LIN {X 0,Y 518.643,Z 984.893,A -85,B 0,C 180,E1 13734.42,E2 13734.42} C_VEL
LIN {X 0,Y 513.947,Z 1023.237,A -85,B 0,C 180,E1 13735.843,E2 13735.843} C_VEL
LIN {X 0,Y 507.593,Z 1061.404,A -85,B 0,C 180,E1 13737.996,E2 13737.996} C_VEL
LIN {X 0,Y 500.506,Z 1096.206,A -85,B 0,C 180,E1 13740.779,E2 13740.779} C_VEL
LIN {X 0,Y 493.713,Z 1126.296,A -85,B 0,C 180,E1 13744.065,E2 13744.065} C_VEL
LIN {X 0,Y 487.682,Z 1152.198,A -85,B 0,C 180,E1 13747.868,E2 13747.868} C_VEL
LIN {X 0,Y 482.961,Z 1173.823,A -85,B 0,C 180,E1 13752.188,E2 13752.188} C_VEL
LIN {X 0,Y 479.947,Z 1190.195,A -85,B 0,C 180,E1 13756.768,E2 13756.768} C_VEL
LIN {X 0,Y 478.377,Z 1201.901,A -85,B 0,C 180,E1 13761.805,E2 13761.805} C_VEL
LIN {X 0,Y 477.916,Z 1207.569,A -85,B 0,C 180,E1 13766.365,E2 13766.365} C_VEL
LIN {X 0,Y 477.819,Z 1208.936,A -85,B 0,C 180,E1 13770,E2 13770} C_VEL
LIN {X 0,Y 477.91,Z 1207.483,A -85,B 0,C 180,E1 13773.636,E2 13773.636} C_VEL
LIN {X 0,Y 478.43,Z 1201.745,A -85,B 0,C 180,E1 13778.194,E2 13778.194} C_VEL
LIN {X 0,Y 480,Z 1189.926,A -85,B 0,C 180,E1 13783.231,E2 13783.231} C_VEL
LIN {X 0,Y 483.195,Z 1172.465,A -85,B 0,C 180,E1 13788.04,E2 13788.04} C_VEL
LIN {X 0,Y 488.136,Z 1150.333,A -85,B 0,C 180,E1 13792.351,E2 13792.351} C_VEL
LIN {X 0,Y 494.263,Z 1123.856,A -85,B 0,C 180,E1 13796.149,E2 13796.149} C_VEL
LIN {X 0,Y 501.436,Z 1091.752,A -85,B 0,C 180,E1 13799.535,E2 13799.535} C_VEL
LIN {X 0,Y 508.377,Z 1056.676,A -85,B 0,C 180,E1 13802.222,E2 13802.222} C_VEL
LIN {X 0,Y 514.491,Z 1018.573,A -85,B 0,C 180,E1 13804.271,E2 13804.271} C_VEL
LIN {X 0,Y 519.025,Z 979.497,A -85,B 0,C 180,E1 13805.64,E2 13805.64} C_VEL
LIN {X 0,Y 520.756,Z 942.856,A -85,B 0,C 180,E1 13806.431,E2 13806.431} C_VEL
LIN {X 0,Y 499.338,Z 900.262,A -85,B 0,C 180,E1 13809.238,E2 13809.238} C_VEL
LIN {X 0,Y 477.541,Z 863.723,A -85,B 0,C 180,E1 13812.378,E2 13812.378} C_VEL
LIN {X 0,Y 476.202,Z 859.31,A -85,B 0,C 180,E1 13812.759,E2 13812.759} C_VEL
LIN {X 0,Y 476.028,Z 859.31,A -85,B 0,C 180,E1 13819.816,E2 13819.816} C_VEL
LIN {X 0,Y 476.22,Z 859.31,A -85,B 0,C 180,E1 13825.823,E2 13825.823} C_VEL
LIN {X 0,Y 476.377,Z 859.31,A -85,B 0,C 180,E1 13831.513,E2 13831.513} C_VEL
LIN {X 0,Y 476.557,Z 859.31,A -85,B 0,C 180,E1 13837.579,E2 13837.579} C_VEL
LIN {X 0,Y 476.651,Z 859.31,A -85,B 0,C 180,E1 13843.382,E2 13843.382} C_VEL
LIN {X 0,Y 477.094,Z 859.31,A -85,B 0,C 180,E1 13849.929,E2 13849.929} C_VEL
LIN {X 0,Y 477.532,Z 859.31,A -85,B 0,C 180,E1 13856.365,E2 13856.365} C_VEL
LIN {X 0,Y 477.649,Z 859.31,A -85,B 0,C 180,E1 13861.82,E2 13861.82} C_VEL
LIN {X 0,Y 477.243,Z 859.31,A -85,B 0,C 180,E1 13867.297,E2 13867.297} C_VEL
LIN {X 0,Y 476.971,Z 859.31,A -85,B 0,C 180,E1 13872.848,E2 13872.848} C_VEL
LIN {X 0,Y 476.774,Z 859.31,A -85,B 0,C 180,E1 13878.529,E2 13878.529} C_VEL
LIN {X 0,Y 476.542,Z 859.31,A -85,B 0,C 180,E1 13884.412,E2 13884.412} C_VEL
LIN {X 0,Y 476.279,Z 859.31,A -85,B 0,C 180,E1 13890.794,E2 13890.794} C_VEL
LIN {X 0,Y 476.088,Z 859.31,A -85,B 0,C 180,E1 13897.278,E2 13897.278} C_VEL
LIN {X 0,Y 476.085,Z 859.334,A -85,B 0,C 180,E1 13901.129,E2 13901.129} C_VEL
LIN {X 0,Y 478.529,Z 865.012,A -85,B 0,C 180,E1 13901.556,E2 13901.556} C_VEL
LIN {X 0,Y 502.826,Z 908.11,A -85,B 0,C 180,E1 13905.163,E2 13905.163} C_VEL
LIN {X 0,Y 518.318,Z 943.312,A -85,B 0,C 180,E1 13907.539,E2 13907.539} C_VEL
LIN {X 0,Y 520.224,Z 951.642,A -85,B 0,C 180,E1 13908,E2 13908} C_VEL
LIN {X 0,Y 515.804,Z 993.529,A -85,B 0,C 180,E1 13909.437,E2 13909.437} C_VEL
LIN {X 0,Y 509.794,Z 1036.666,A -85,B 0,C 180,E1 13911.635,E2 13911.635} C_VEL
LIN {X 0,Y 502.567,Z 1078.417,A -85,B 0,C 180,E1 13914.594,E2 13914.594} C_VEL
LIN {X 0,Y 495.342,Z 1116.789,A -85,B 0,C 180,E1 13918.279,E2 13918.279} C_VEL
LIN {X 0,Y 488.813,Z 1150.319,A -85,B 0,C 180,E1 13922.541,E2 13922.541} C_VEL
LIN {X 0,Y 483.649,Z 1178.839,A -85,B 0,C 180,E1 13927.341,E2 13927.341} C_VEL
LIN {X 0,Y 480.223,Z 1201.767,A -85,B 0,C 180,E1 13932.556,E2 13932.556} C_VEL
LIN {X 0,Y 478.57,Z 1217.65,A -85,B 0,C 180,E1 13937.659,E2 13937.659} C_VEL
LIN {X 0,Y 477.922,Z 1227.864,A -85,B 0,C 180,E1 13942.714,E2 13942.714} C_VEL
LIN {X 0,Y 477.728,Z 1232.511,A -85,B 0,C 180,E1 13947.322,E2 13947.322} C_VEL
LIN {X 0,Y 475.241,Z 1233.109,A -85,B 0,C 180,E1 13948.872,E2 13948.872} C_VEL
LIN {X 0,Y 469.933,Z 1232.933,A -85,B 0,C 180,E1 13951.202,E2 13951.202} C_VEL
LIN {X 0,Y 469.852,Z 1232.873,A -85,B 0,C 180,E1 13951.471,E2 13951.471} C_VEL
LIN {X 0,Y 470.024,Z 1228.932,A -85,B 0,C 180,E1 13956.479,E2 13956.479} C_VEL
LIN {X 0,Y 470.546,Z 1219.738,A -85,B 0,C 180,E1 13961.611,E2 13961.611} C_VEL
LIN {X 0,Y 472.095,Z 1204.807,A -85,B 0,C 180,E1 13966.79,E2 13966.79} C_VEL
LIN {X 0,Y 475.116,Z 1184.672,A -85,B 0,C 180,E1 13971.762,E2 13971.762} C_VEL
LIN {X 0,Y 479.783,Z 1159.104,A -85,B 0,C 180,E1 13976.494,E2 13976.494} C_VEL
LIN {X 0,Y 486.088,Z 1127.252,A -85,B 0,C 180,E1 13980.964,E2 13980.964} C_VEL
LIN {X 0,Y 493.608,Z 1090.252,A -85,B 0,C 180,E1 13984.873,E2 13984.873} C_VEL
LIN {X 0,Y 501.082,Z 1049.955,A -85,B 0,C 180,E1 13988.053,E2 13988.053} C_VEL
LIN {X 0,Y 507.902,Z 1006.301,A -85,B 0,C 180,E1 13990.547,E2 13990.547} C_VEL
LIN {X 0,Y 513.509,Z 959.069,A -85,B 0,C 180,E1 13992.355,E2 13992.355} C_VEL
LIN {X 0,Y 513.392,Z 950.47,A -85,B 0,C 180,E1 13992.673,E2 13992.673} C_VEL
LIN {X 0,Y 500.582,Z 918.482,A -85,B 0,C 180,E1 13994.85,E2 13994.85} C_VEL
LIN {X 0,Y 477.749,Z 876.402,A -85,B 0,C 180,E1 13998.301,E2 13998.301} C_VEL
LIN {X 0,Y 468.278,Z 860.452,A -85,B 0,C 180,E1 13999.854,E2 13999.854} C_VEL
LIN {X 0,Y 468.166,Z 859.31,A -85,B 0,C 180,E1 14000.015,E2 14000.015} C_VEL
LIN {X 0,Y 468.263,Z 859.31,A -85,B 0,C 180,E1 14006.632,E2 14006.632} C_VEL
LIN {X 0,Y 468.524,Z 859.31,A -85,B 0,C 180,E1 14013.082,E2 14013.082} C_VEL
LIN {X 0,Y 468.832,Z 859.31,A -85,B 0,C 180,E1 14019.602,E2 14019.602} C_VEL
LIN {X 0,Y 468.939,Z 859.31,A -85,B 0,C 180,E1 14025.787,E2 14025.787} C_VEL
LIN {X 0,Y 469.249,Z 859.31,A -85,B 0,C 180,E1 14030.708,E2 14030.708} C_VEL
LIN {X 0,Y 469.615,Z 859.31,A -85,B 0,C 180,E1 14036.298,E2 14036.298} C_VEL
LIN {X 0,Y 469.762,Z 859.31,A -85,B 0,C 180,E1 14041.845,E2 14041.845} C_VEL
LIN {X 0,Y 469.331,Z 859.31,A -85,B 0,C 180,E1 14047.416,E2 14047.416} C_VEL
LIN {X 0,Y 469.047,Z 859.31,A -85,B 0,C 180,E1 14053.064,E2 14053.064} C_VEL
LIN {X 0,Y 468.807,Z 859.31,A -85,B 0,C 180,E1 14058.85,E2 14058.85} C_VEL
LIN {X 0,Y 468.505,Z 859.31,A -85,B 0,C 180,E1 14065.095,E2 14065.095} C_VEL
LIN {X 0,Y 468.309,Z 859.31,A -85,B 0,C 180,E1 14071.166,E2 14071.166} C_VEL
LIN {X 0,Y 468.114,Z 859.31,A -85,B 0,C 180,E1 14077.939,E2 14077.939} C_VEL
LIN {X 0,Y 468.115,Z 859.31,A -85,B 0,C 180,E1 14084.591,E2 14084.591} C_VEL
LIN {X 0,Y 468.174,Z 859.802,A -85,B 0,C 180,E1 14086.245,E2 14086.245} C_VEL
LIN {X 0,Y 470.923,Z 865.256,A -85,B 0,C 180,E1 14086.71,E2 14086.71} C_VEL
LIN {X 0,Y 495.158,Z 906.292,A -85,B 0,C 180,E1 14090.317,E2 14090.317} C_VEL
LIN {X 0,Y 515.205,Z 946.752,A -85,B 0,C 180,E1 14093.03,E2 14093.03} C_VEL
LIN {X 0,Y 512.18,Z 987.401,A -85,B 0,C 180,E1 14093.945,E2 14093.945} C_VEL
LIN {X 0,Y 507.237,Z 1025.551,A -85,B 0,C 180,E1 14095.418,E2 14095.418} C_VEL
LIN {X 0,Y 500.822,Z 1062.523,A -85,B 0,C 180,E1 14097.556,E2 14097.556} C_VEL
LIN {X 0,Y 493.611,Z 1096.638,A -85,B 0,C 180,E1 14100.33,E2 14100.33} C_VEL
LIN {X 0,Y 486.56,Z 1126.639,A -85,B 0,C 180,E1 14103.654,E2 14103.654} C_VEL
LIN {X 0,Y 480.259,Z 1152.487,A -85,B 0,C 180,E1 14107.508,E2 14107.508} C_VEL
LIN {X 0,Y 475.347,Z 1174.075,A -85,B 0,C 180,E1 14111.892,E2 14111.892} C_VEL
LIN {X 0,Y 472.183,Z 1190.422,A -85,B 0,C 180,E1 14116.546,E2 14116.546} C_VEL
LIN {X 0,Y 470.51,Z 1202.111,A -85,B 0,C 180,E1 14121.667,E2 14121.667} C_VEL
LIN {X 0,Y 470.017,Z 1207.774,A -85,B 0,C 180,E1 14126.303,E2 14126.303} C_VEL
LIN {X 0,Y 469.922,Z 1209.138,A -85,B 0,C 180,E1 14130,E2 14130} C_VEL
LIN {X 0,Y 470.013,Z 1207.688,A -85,B 0,C 180,E1 14133.697,E2 14133.697} C_VEL
LIN {X 0,Y 470.558,Z 1201.957,A -85,B 0,C 180,E1 14138.332,E2 14138.332} C_VEL
LIN {X 0,Y 472.233,Z 1190.156,A -85,B 0,C 180,E1 14143.453,E2 14143.453} C_VEL
LIN {X 0,Y 475.608,Z 1172.733,A -85,B 0,C 180,E1 14148.338,E2 14148.338} C_VEL
LIN {X 0,Y 481.056,Z 1149.238,A -85,B 0,C 180,E1 14152.943,E2 14152.943} C_VEL
LIN {X 0,Y 487.547,Z 1122.37,A -85,B 0,C 180,E1 14156.786,E2 14156.786} C_VEL
LIN {X 0,Y 494.822,Z 1090.999,A -85,B 0,C 180,E1 14160.096,E2 14160.096} C_VEL
LIN {X 0,Y 501.843,Z 1056.834,A -85,B 0,C 180,E1 14162.732,E2 14162.732} C_VEL
LIN {X 0,Y 508.188,Z 1018.409,A -85,B 0,C 180,E1 14164.819,E2 14164.819} C_VEL
LIN {X 0,Y 512.975,Z 978.573,A -85,B 0,C 180,E1 14166.213,E2 14166.213} C_VEL
LIN {X 0,Y 514.693,Z 945.644,A -85,B 0,C 180,E1 14166.937,E2 14166.937} C_VEL
LIN {X 0,Y 492.273,Z 901.174,A -85,B 0,C 180,E1 14169.979,E2 14169.979} C_VEL
LIN {X 0,Y 470.238,Z 864.606,A -85,B 0,C 180,E1 14173.277,E2 14173.277} C_VEL
LIN {X 0,Y 468.154,Z 859.31,A -85,B 0,C 180,E1 14173.753,E2 14173.753} C_VEL
LIN {X 0,Y 468.127,Z 859.31,A -85,B 0,C 180,E1 14179.672,E2 14179.672} C_VEL
LIN {X 0,Y 468.287,Z 859.31,A -85,B 0,C 180,E1 14186.64,E2 14186.64} C_VEL
LIN {X 0,Y 468.477,Z 859.31,A -85,B 0,C 180,E1 14193.085,E2 14193.085} C_VEL
LIN {X 0,Y 468.671,Z 859.31,A -85,B 0,C 180,E1 14199.656,E2 14199.656} C_VEL
LIN {X 0,Y 468.844,Z 859.31,A -85,B 0,C 180,E1 14205.836,E2 14205.836} C_VEL
LIN {X 0,Y 469.33,Z 859.31,A -85,B 0,C 180,E1 14212.227,E2 14212.227} C_VEL
LIN {X 0,Y 469.667,Z 859.31,A -85,B 0,C 180,E1 14218.154,E2 14218.154} C_VEL
LIN {X 0,Y 469.601,Z 859.31,A -85,B 0,C 180,E1 14223.702,E2 14223.702} C_VEL
LIN {X 0,Y 469.229,Z 859.31,A -85,B 0,C 180,E1 14229.292,E2 14229.292} C_VEL
LIN {X 0,Y 468.986,Z 859.31,A -85,B 0,C 180,E1 14234.978,E2 14234.978} C_VEL
LIN {X 0,Y 468.782,Z 859.31,A -85,B 0,C 180,E1 14240.825,E2 14240.825} C_VEL
LIN {X 0,Y 468.497,Z 859.31,A -85,B 0,C 180,E1 14246.919,E2 14246.919} C_VEL
LIN {X 0,Y 468.277,Z 859.31,A -85,B 0,C 180,E1 14253.367,E2 14253.367} C_VEL
LIN {X 0,Y 468.111,Z 859.312,A -85,B 0,C 180,E1 14260.118,E2 14260.118} C_VEL
LIN {X 0,Y 470.283,Z 864.719,A -85,B 0,C 180,E1 14260.525,E2 14260.525} C_VEL
LIN {X 0,Y 492.086,Z 902.116,A -85,B 0,C 180,E1 14263.914,E2 14263.914} C_VEL
LIN {X 0,Y 509.924,Z 939.992,A -85,B 0,C 180,E1 14266.663,E2 14266.663} C_VEL
LIN {X 0,Y 513.917,Z 953.77,A -85,B 0,C 180,E1 14267.504,E2 14267.504} C_VEL
LIN {X 0,Y 509.349,Z 994.883,A -85,B 0,C 180,E1 14268.95,E2 14268.95} C_VEL
LIN {X 0,Y 503.273,Z 1036.889,A -85,B 0,C 180,E1 14271.119,E2 14271.119} C_VEL
LIN {X 0,Y 495.963,Z 1077.869,A -85,B 0,C 180,E1 14274.05,E2 14274.05} C_VEL
LIN {X 0,Y 488.496,Z 1115.732,A -85,B 0,C 180,E1 14277.704,E2 14277.704} C_VEL
LIN {X 0,Y 481.527,Z 1149.949,A -85,B 0,C 180,E1 14282.089,E2 14282.089} C_VEL
LIN {X 0,Y 476.023,Z 1178.977,A -85,B 0,C 180,E1 14287.05,E2 14287.05} C_VEL
LIN {X 0,Y 472.472,Z 1201.489,A -85,B 0,C 180,E1 14292.261,E2 14292.261} C_VEL
LIN {X 0,Y 470.711,Z 1217.409,A -85,B 0,C 180,E1 14297.45,E2 14297.45} C_VEL
LIN {X 0,Y 470.105,Z 1226.204,A -85,B 0,C 180,E1 14301.66,E2 14301.66} C_VEL
LIN {X 0,Y 469.844,Z 1231.759,A -85,B 0,C 180,E1 14306.302,E2 14306.302} C_VEL
LIN {X 0,Y 469.936,Z 1233.157,A -85,B 0,C 180,E1 14310,E2 14310} C_VEL
LIN {X 0,Y 469.852,Z 1232.873,A -85,B 0,C 180,E1 14311.471,E2 14311.471} C_VEL
LIN {X 0,Y 467.415,Z 1232.232,A -85,B 0,C 180,E1 14313.044,E2 14313.044} C_VEL
LIN {X 0,Y 462.169,Z 1230.135,A -85,B 0,C 180,E1 14315.394,E2 14315.394} C_VEL
LIN {X 0,Y 462.077,Z 1229.821,A -85,B 0,C 180,E1 14315.664,E2 14315.664} C_VEL
LIN {X 0,Y 462.495,Z 1221.924,A -85,B 0,C 180,E1 14320.678,E2 14320.678} C_VEL
LIN {X 0,Y 463.939,Z 1207.878,A -85,B 0,C 180,E1 14326.085,E2 14326.085} C_VEL
LIN {X 0,Y 467.146,Z 1186.79,A -85,B 0,C 180,E1 14331.62,E2 14331.62} C_VEL
LIN {X 0,Y 472.159,Z 1160.263,A -85,B 0,C 180,E1 14336.699,E2 14336.699} C_VEL
LIN {X 0,Y 478.842,Z 1128.024,A -85,B 0,C 180,E1 14341.325,E2 14341.325} C_VEL
LIN {X 0,Y 486.665,Z 1091.024,A -85,B 0,C 180,E1 14345.307,E2 14345.307} C_VEL
LIN {X 0,Y 494.453,Z 1050.57,A -85,B 0,C 180,E1 14348.549,E2 14348.549} C_VEL
LIN {X 0,Y 501.632,Z 1006.288,A -85,B 0,C 180,E1 14351.104,E2 14351.104} C_VEL
LIN {X 0,Y 507.368,Z 959.498,A -85,B 0,C 180,E1 14352.911,E2 14352.911} C_VEL
LIN {X 0,Y 506.856,Z 951.867,A -85,B 0,C 180,E1 14353.238,E2 14353.238} C_VEL
LIN {X 0,Y 492.383,Z 916.889,A -85,B 0,C 180,E1 14355.747,E2 14355.747} C_VEL
LIN {X 0,Y 470.309,Z 876.985,A -85,B 0,C 180,E1 14359.208,E2 14359.208} C_VEL
LIN {X 0,Y 460.437,Z 860.936,A -85,B 0,C 180,E1 14360.89,E2 14360.89} C_VEL
LIN {X 0,Y 460.251,Z 859.31,A -85,B 0,C 180,E1 14361.01,E2 14361.01} C_VEL
LIN {X 0,Y 460.401,Z 859.31,A -85,B 0,C 180,E1 14368.23,E2 14368.23} C_VEL
LIN {X 0,Y 460.636,Z 859.31,A -85,B 0,C 180,E1 14374.686,E2 14374.686} C_VEL
LIN {X 0,Y 460.894,Z 859.31,A -85,B 0,C 180,E1 14380.808,E2 14380.808} C_VEL
LIN {X 0,Y 461.078,Z 859.31,A -85,B 0,C 180,E1 14386.701,E2 14386.701} C_VEL
LIN {X 0,Y 461.42,Z 859.31,A -85,B 0,C 180,E1 14392.451,E2 14392.451} C_VEL
LIN {X 0,Y 461.757,Z 859.31,A -85,B 0,C 180,E1 14398.117,E2 14398.117} C_VEL
LIN {X 0,Y 461.683,Z 859.31,A -85,B 0,C 180,E1 14403.76,E2 14403.76} C_VEL
LIN {X 0,Y 461.272,Z 859.31,A -85,B 0,C 180,E1 14409.767,E2 14409.767} C_VEL
LIN {X 0,Y 461.038,Z 859.31,A -85,B 0,C 180,E1 14415.238,E2 14415.238} C_VEL
LIN {X 0,Y 460.793,Z 859.31,A -85,B 0,C 180,E1 14421.198,E2 14421.198} C_VEL
LIN {X 0,Y 460.495,Z 859.31,A -85,B 0,C 180,E1 14427.42,E2 14427.42} C_VEL
LIN {X 0,Y 460.392,Z 859.31,A -85,B 0,C 180,E1 14431.764,E2 14431.764} C_VEL
LIN {X 0,Y 460.187,Z 859.31,A -85,B 0,C 180,E1 14438.713,E2 14438.713} C_VEL
LIN {X 0,Y 460.214,Z 859.407,A -85,B 0,C 180,E1 14445.165,E2 14445.165} C_VEL
LIN {X 0,Y 462.529,Z 864.884,A -85,B 0,C 180,E1 14445.597,E2 14445.597} C_VEL
LIN {X 0,Y 484.481,Z 900.745,A -85,B 0,C 180,E1 14449.032,E2 14449.032} C_VEL
LIN {X 0,Y 506.711,Z 944.18,A -85,B 0,C 180,E1 14452.164,E2 14452.164} C_VEL
LIN {X 0,Y 509.1,Z 950.401,A -85,B 0,C 180,E1 14452.522,E2 14452.522} C_VEL
LIN {X 0,Y 505.553,Z 991.888,A -85,B 0,C 180,E1 14453.521,E2 14453.521} C_VEL
LIN {X 0,Y 500.14,Z 1030.636,A -85,B 0,C 180,E1 14455.12,E2 14455.12} C_VEL
LIN {X 0,Y 493.483,Z 1066.438,A -85,B 0,C 180,E1 14457.302,E2 14457.302} C_VEL
LIN {X 0,Y 486.19,Z 1099.316,A -85,B 0,C 180,E1 14460.088,E2 14460.088} C_VEL
LIN {X 0,Y 478.994,Z 1128.68,A -85,B 0,C 180,E1 14463.459,E2 14463.459} C_VEL
LIN {X 0,Y 472.565,Z 1154.05,A -85,B 0,C 180,E1 14467.37,E2 14467.37} C_VEL
LIN {X 0,Y 467.733,Z 1174.324,A -85,B 0,C 180,E1 14471.587,E2 14471.587} C_VEL
LIN {X 0,Y 464.447,Z 1190.646,A -85,B 0,C 180,E1 14476.318,E2 14476.318} C_VEL
LIN {X 0,Y 462.645,Z 1202.321,A -85,B 0,C 180,E1 14481.525,E2 14481.525} C_VEL
LIN {X 0,Y 462.119,Z 1207.978,A -85,B 0,C 180,E1 14486.24,E2 14486.24} C_VEL
LIN {X 0,Y 462.039,Z 1209.339,A -85,B 0,C 180,E1 14490,E2 14490} C_VEL
LIN {X 0,Y 462.116,Z 1207.894,A -85,B 0,C 180,E1 14493.76,E2 14493.76} C_VEL
LIN {X 0,Y 462.691,Z 1202.168,A -85,B 0,C 180,E1 14498.475,E2 14498.475} C_VEL
LIN {X 0,Y 464.494,Z 1190.383,A -85,B 0,C 180,E1 14503.681,E2 14503.681} C_VEL
LIN {X 0,Y 467.779,Z 1173.951,A -85,B 0,C 180,E1 14508.411,E2 14508.411} C_VEL
LIN {X 0,Y 473.371,Z 1150.953,A -85,B 0,C 180,E1 14513.087,E2 14513.087} C_VEL
LIN {X 0,Y 480.447,Z 1122.744,A -85,B 0,C 180,E1 14517.215,E2 14517.215} C_VEL
LIN {X 0,Y 487.993,Z 1091.476,A -85,B 0,C 180,E1 14520.562,E2 14520.562} C_VEL
LIN {X 0,Y 495.345,Z 1057.016,A -85,B 0,C 180,E1 14523.253,E2 14523.253} C_VEL
LIN {X 0,Y 501.866,Z 1018.788,A -85,B 0,C 180,E1 14525.355,E2 14525.355} C_VEL
LIN {X 0,Y 506.858,Z 978.632,A -85,B 0,C 180,E1 14526.777,E2 14526.777} C_VEL
LIN {X 0,Y 508.419,Z 948.038,A -85,B 0,C 180,E1 14527.487,E2 14527.487} C_VEL
LIN {X 0,Y 487.116,Z 905.608,A -85,B 0,C 180,E1 14530.471,E2 14530.471} C_VEL
LIN {X 0,Y 465.526,Z 869.667,A -85,B 0,C 180,E1 14533.79,E2 14533.79} C_VEL
LIN {X 0,Y 460.319,Z 860.503,A -85,B 0,C 180,E1 14534.68,E2 14534.68} C_VEL
LIN {X 0,Y 460.225,Z 859.31,A -85,B 0,C 180,E1 14534.724,E2 14534.724} C_VEL
LIN {X 0,Y 460.213,Z 859.31,A -85,B 0,C 180,E1 14541.29,E2 14541.29} C_VEL
LIN {X 0,Y 460.4,Z 859.31,A -85,B 0,C 180,E1 14548.236,E2 14548.236} C_VEL
LIN {X 0,Y 460.585,Z 859.31,A -85,B 0,C 180,E1 14554.689,E2 14554.689} C_VEL
LIN {X 0,Y 460.732,Z 859.31,A -85,B 0,C 180,E1 14560.807,E2 14560.807} C_VEL
LIN {X 0,Y 461.022,Z 859.31,A -85,B 0,C 180,E1 14566.705,E2 14566.705} C_VEL
LIN {X 0,Y 461.463,Z 859.31,A -85,B 0,C 180,E1 14572.457,E2 14572.457} C_VEL
LIN {X 0,Y 461.762,Z 859.31,A -85,B 0,C 180,E1 14578.123,E2 14578.123} C_VEL
LIN {X 0,Y 461.688,Z 859.31,A -85,B 0,C 180,E1 14583.765,E2 14583.765} C_VEL
LIN {X 0,Y 461.264,Z 859.31,A -85,B 0,C 180,E1 14589.759,E2 14589.759} C_VEL
LIN {X 0,Y 461.045,Z 859.31,A -85,B 0,C 180,E1 14595.243,E2 14595.243} C_VEL
LIN {X 0,Y 460.823,Z 859.31,A -85,B 0,C 180,E1 14601.202,E2 14601.202} C_VEL
LIN {X 0,Y 460.52,Z 859.31,A -85,B 0,C 180,E1 14607.424,E2 14607.424} C_VEL
LIN {X 0,Y 460.408,Z 859.31,A -85,B 0,C 180,E1 14611.769,E2 14611.769} C_VEL
LIN {X 0,Y 460.217,Z 859.31,A -85,B 0,C 180,E1 14618.991,E2 14618.991} C_VEL
LIN {X 0,Y 462.795,Z 865.147,A -85,B 0,C 180,E1 14619.555,E2 14619.555} C_VEL
LIN {X 0,Y 484.819,Z 902.715,A -85,B 0,C 180,E1 14623.122,E2 14623.122} C_VEL
LIN {X 0,Y 502.161,Z 938.918,A -85,B 0,C 180,E1 14625.876,E2 14625.876} C_VEL
LIN {X 0,Y 507.634,Z 956.314,A -85,B 0,C 180,E1 14627.01,E2 14627.01} C_VEL
LIN {X 0,Y 502.713,Z 998.007,A -85,B 0,C 180,E1 14628.531,E2 14628.531} C_VEL
LIN {X 0,Y 496.473,Z 1038.942,A -85,B 0,C 180,E1 14630.707,E2 14630.707} C_VEL
LIN {X 0,Y 488.925,Z 1079.443,A -85,B 0,C 180,E1 14633.671,E2 14633.671} C_VEL
LIN {X 0,Y 481.158,Z 1117.321,A -85,B 0,C 180,E1 14637.415,E2 14637.415} C_VEL
LIN {X 0,Y 473.962,Z 1151.139,A -85,B 0,C 180,E1 14641.864,E2 14641.864} C_VEL
LIN {X 0,Y 468.524,Z 1178.663,A -85,B 0,C 180,E1 14646.66,E2 14646.66} C_VEL
LIN {X 0,Y 464.735,Z 1201.218,A -85,B 0,C 180,E1 14651.955,E2 14651.955} C_VEL
LIN {X 0,Y 462.873,Z 1217.171,A -85,B 0,C 180,E1 14657.234,E2 14657.234} C_VEL
LIN {X 0,Y 462.216,Z 1225.984,A -85,B 0,C 180,E1 14661.516,E2 14661.516} C_VEL
LIN {X 0,Y 461.942,Z 1231.555,A -85,B 0,C 180,E1 14666.238,E2 14666.238} C_VEL
LIN {X 0,Y 462.055,Z 1232.956,A -85,B 0,C 180,E1 14670,E2 14670} C_VEL
LIN {X 0,Y 462.003,Z 1231.559,A -85,B 0,C 180,E1 14673.761,E2 14673.761} C_VEL
LIN {X 0,Y 462.077,Z 1229.821,A -85,B 0,C 180,E1 14675.664,E2 14675.664} C_VEL
LIN {X 0,Y 460.831,Z 1228.526,A -85,B 0,C 180,E1 14676.726,E2 14676.726} C_VEL
LIN {X 0,Y 454.504,Z 1224.099,A -85,B 0,C 180,E1 14679.609,E2 14679.609} C_VEL
LIN {X 0,Y 454.462,Z 1223.629,A -85,B 0,C 180,E1 14679.881,E2 14679.881} C_VEL
LIN {X 0,Y 455.613,Z 1211.823,A -85,B 0,C 180,E1 14684.936,E2 14684.936} C_VEL
LIN {X 0,Y 458.186,Z 1193.554,A -85,B 0,C 180,E1 14690.319,E2 14690.319} C_VEL
LIN {X 0,Y 462.843,Z 1169.569,A -85,B 0,C 180,E1 14695.455,E2 14695.455} C_VEL
LIN {X 0,Y 469.331,Z 1139.313,A -85,B 0,C 180,E1 14700.296,E2 14700.296} C_VEL
LIN {X 0,Y 477.217,Z 1103.192,A -85,B 0,C 180,E1 14704.629,E2 14704.629} C_VEL
LIN {X 0,Y 485.591,Z 1063.104,A -85,B 0,C 180,E1 14708.188,E2 14708.188} C_VEL
LIN {X 0,Y 493.207,Z 1020.517,A -85,B 0,C 180,E1 14710.946,E2 14710.946} C_VEL
LIN {X 0,Y 499.618,Z 975.313,A -85,B 0,C 180,E1 14712.967,E2 14712.967} C_VEL
LIN {X 0,Y 501.077,Z 955.78,A -85,B 0,C 180,E1 14713.655,E2 14713.655} C_VEL
LIN {X 0,Y 487.368,Z 921.772,A -85,B 0,C 180,E1 14716.172,E2 14716.172} C_VEL
LIN {X 0,Y 466.105,Z 882.842,A -85,B 0,C 180,E1 14719.61,E2 14719.61} C_VEL
LIN {X 0,Y 452.501,Z 860.973,A -85,B 0,C 180,E1 14722.009,E2 14722.009} C_VEL
LIN {X 0,Y 452.314,Z 859.31,A -85,B 0,C 180,E1 14722.178,E2 14722.178} C_VEL
LIN {X 0,Y 452.388,Z 859.31,A -85,B 0,C 180,E1 14727.6,E2 14727.6} C_VEL
LIN {X 0,Y 452.669,Z 859.31,A -85,B 0,C 180,E1 14734.208,E2 14734.208} C_VEL
LIN {X 0,Y 452.941,Z 859.31,A -85,B 0,C 180,E1 14740.458,E2 14740.458} C_VEL
LIN {X 0,Y 453.14,Z 859.31,A -85,B 0,C 180,E1 14746.464,E2 14746.464} C_VEL
LIN {X 0,Y 453.51,Z 859.31,A -85,B 0,C 180,E1 14752.319,E2 14752.319} C_VEL
LIN {X 0,Y 453.875,Z 859.31,A -85,B 0,C 180,E1 14758.085,E2 14758.085} C_VEL
LIN {X 0,Y 453.778,Z 859.31,A -85,B 0,C 180,E1 14763.826,E2 14763.826} C_VEL
LIN {X 0,Y 453.403,Z 859.31,A -85,B 0,C 180,E1 14769.614,E2 14769.614} C_VEL
LIN {X 0,Y 453.111,Z 859.31,A -85,B 0,C 180,E1 14775.511,E2 14775.511} C_VEL
LIN {X 0,Y 452.855,Z 859.31,A -85,B 0,C 180,E1 14781.588,E2 14781.588} C_VEL
LIN {X 0,Y 452.52,Z 859.31,A -85,B 0,C 180,E1 14787.945,E2 14787.945} C_VEL
LIN {X 0,Y 452.337,Z 859.31,A -85,B 0,C 180,E1 14794.701,E2 14794.701} C_VEL
LIN {X 0,Y 452.218,Z 859.31,A -85,B 0,C 180,E1 14799.585,E2 14799.585} C_VEL
LIN {X 0,Y 452.293,Z 859.31,A -85,B 0,C 180,E1 14804.002,E2 14804.002} C_VEL
LIN {X 0,Y 454.772,Z 865.018,A -85,B 0,C 180,E1 14804.52,E2 14804.52} C_VEL
LIN {X 0,Y 476.117,Z 899.474,A -85,B 0,C 180,E1 14808.024,E2 14808.024} C_VEL
LIN {X 0,Y 497.352,Z 939.652,A -85,B 0,C 180,E1 14811.13,E2 14811.13} C_VEL
LIN {X 0,Y 502.965,Z 952.207,A -85,B 0,C 180,E1 14811.958,E2 14811.958} C_VEL
LIN {X 0,Y 498.971,Z 995.969,A -85,B 0,C 180,E1 14813.079,E2 14813.079} C_VEL
LIN {X 0,Y 493.057,Z 1035.538,A -85,B 0,C 180,E1 14814.814,E2 14814.814} C_VEL
LIN {X 0,Y 485.711,Z 1072.495,A -85,B 0,C 180,E1 14817.211,E2 14817.211} C_VEL
LIN {X 0,Y 477.815,Z 1105.983,A -85,B 0,C 180,E1 14820.256,E2 14820.256} C_VEL
LIN {X 0,Y 470.14,Z 1135.582,A -85,B 0,C 180,E1 14823.938,E2 14823.938} C_VEL
LIN {X 0,Y 463.631,Z 1160.578,A -85,B 0,C 180,E1 14828.175,E2 14828.175} C_VEL
LIN {X 0,Y 458.922,Z 1180.103,A -85,B 0,C 180,E1 14832.713,E2 14832.713} C_VEL
LIN {X 0,Y 455.787,Z 1195.793,A -85,B 0,C 180,E1 14838.008,E2 14838.008} C_VEL
LIN {X 0,Y 454.496,Z 1205.313,A -85,B 0,C 180,E1 14843.299,E2 14843.299} C_VEL
LIN {X 0,Y 454.136,Z 1209.215,A -85,B 0,C 180,E1 14848.088,E2 14848.088} C_VEL
LIN {X 0,Y 454.247,Z 1209.162,A -85,B 0,C 180,E1 14851.912,E2 14851.912} C_VEL
LIN {X 0,Y 454.525,Z 1205.194,A -85,B 0,C 180,E1 14856.701,E2 14856.701} C_VEL
LIN {X 0,Y 455.85,Z 1195.569,A -85,B 0,C 180,E1 14861.991,E2 14861.991} C_VEL
LIN {X 0,Y 458.951,Z 1179.773,A -85,B 0,C 180,E1 14867.287,E2 14867.287} C_VEL
LIN {X 0,Y 464.04,Z 1158.936,A -85,B 0,C 180,E1 14872.057,E2 14872.057} C_VEL
LIN {X 0,Y 470.756,Z 1133.212,A -85,B 0,C 180,E1 14876.306,E2 14876.306} C_VEL
LIN {X 0,Y 478.443,Z 1103.378,A -85,B 0,C 180,E1 14879.92,E2 14879.92} C_VEL
LIN {X 0,Y 486.284,Z 1069.61,A -85,B 0,C 180,E1 14882.911,E2 14882.911} C_VEL
LIN {X 0,Y 493.562,Z 1031.945,A -85,B 0,C 180,E1 14885.28,E2 14885.28} C_VEL
LIN {X 0,Y 499.328,Z 991.839,A -85,B 0,C 180,E1 14886.963,E2 14886.963} C_VEL
LIN {X 0,Y 502.68,Z 951.415,A -85,B 0,C 180,E1 14887.981,E2 14887.981} C_VEL
LIN {X 0,Y 480.79,Z 907.701,A -85,B 0,C 180,E1 14891.155,E2 14891.155} C_VEL
LIN {X 0,Y 458.577,Z 870.917,A -85,B 0,C 180,E1 14894.701,E2 14894.701} C_VEL
LIN {X 0,Y 452.499,Z 861.045,A -85,B 0,C 180,E1 14895.776,E2 14895.776} C_VEL
LIN {X 0,Y 452.293,Z 859.31,A -85,B 0,C 180,E1 14895.921,E2 14895.921} C_VEL
LIN {X 0,Y 452.324,Z 859.31,A -85,B 0,C 180,E1 14902.93,E2 14902.93} C_VEL
LIN {X 0,Y 452.519,Z 859.31,A -85,B 0,C 180,E1 14909.861,E2 14909.861} C_VEL
LIN {X 0,Y 452.706,Z 859.31,A -85,B 0,C 180,E1 14916.327,E2 14916.327} C_VEL
LIN {X 0,Y 452.85,Z 859.31,A -85,B 0,C 180,E1 14922.481,E2 14922.481} C_VEL
LIN {X 0,Y 453.23,Z 859.31,A -85,B 0,C 180,E1 14928.434,E2 14928.434} C_VEL
LIN {X 0,Y 453.694,Z 859.31,A -85,B 0,C 180,E1 14934.254,E2 14934.254} C_VEL
LIN {X 0,Y 454.019,Z 859.31,A -85,B 0,C 180,E1 14940.003,E2 14940.003} C_VEL
LIN {X 0,Y 453.69,Z 859.31,A -85,B 0,C 180,E1 14945.752,E2 14945.752} C_VEL
LIN {X 0,Y 453.26,Z 859.31,A -85,B 0,C 180,E1 14951.571,E2 14951.571} C_VEL
LIN {X 0,Y 453.031,Z 859.31,A -85,B 0,C 180,E1 14957.517,E2 14957.517} C_VEL
LIN {X 0,Y 452.773,Z 859.31,A -85,B 0,C 180,E1 14963.675,E2 14963.675} C_VEL
LIN {X 0,Y 452.535,Z 859.31,A -85,B 0,C 180,E1 14970.144,E2 14970.144} C_VEL
LIN {X 0,Y 452.303,Z 859.31,A -85,B 0,C 180,E1 14977.079,E2 14977.079} C_VEL
LIN {X 0,Y 452.311,Z 859.86,A -85,B 0,C 180,E1 14977.96,E2 14977.96} C_VEL
LIN {X 0,Y 455.206,Z 865.447,A -85,B 0,C 180,E1 14978.514,E2 14978.514} C_VEL
LIN {X 0,Y 477.9,Z 903.872,A -85,B 0,C 180,E1 14982.349,E2 14982.349} C_VEL
LIN {X 0,Y 495.693,Z 940.704,A -85,B 0,C 180,E1 14985.276,E2 14985.276} C_VEL
LIN {X 0,Y 501.427,Z 958.119,A -85,B 0,C 180,E1 14986.479,E2 14986.479} C_VEL
LIN {X 0,Y 496.177,Z 1000.576,A -85,B 0,C 180,E1 14988.074,E2 14988.074} C_VEL
LIN {X 0,Y 489.683,Z 1040.936,A -85,B 0,C 180,E1 14990.277,E2 14990.277} C_VEL
LIN {X 0,Y 482.109,Z 1080.122,A -85,B 0,C 180,E1 14993.202,E2 14993.202} C_VEL
LIN {X 0,Y 474.187,Z 1117.166,A -85,B 0,C 180,E1 14996.91,E2 14996.91} C_VEL
LIN {X 0,Y 466.933,Z 1150.061,A -85,B 0,C 180,E1 15001.274,E2 15001.274} C_VEL
LIN {X 0,Y 460.994,Z 1178.355,A -85,B 0,C 180,E1 15006.255,E2 15006.255} C_VEL
LIN {X 0,Y 456.998,Z 1200.95,A -85,B 0,C 180,E1 15011.639,E2 15011.639} C_VEL
LIN {X 0,Y 455.042,Z 1216.936,A -85,B 0,C 180,E1 15017.01,E2 15017.01} C_VEL
LIN {X 0,Y 454.339,Z 1225.765,A -85,B 0,C 180,E1 15021.368,E2 15021.368} C_VEL
LIN {X 0,Y 454.05,Z 1231.35,A -85,B 0,C 180,E1 15026.173,E2 15026.173} C_VEL
LIN {X 0,Y 454.156,Z 1232.754,A -85,B 0,C 180,E1 15030,E2 15030} C_VEL
LIN {X 0,Y 454.099,Z 1231.355,A -85,B 0,C 180,E1 15033.826,E2 15033.826} C_VEL
LIN {X 0,Y 454.295,Z 1225.772,A -85,B 0,C 180,E1 15038.632,E2 15038.632} C_VEL
LIN {X 0,Y 454.462,Z 1223.629,A -85,B 0,C 180,E1 15039.881,E2 15039.881} C_VEL
LIN {X 0,Y 452.246,Z 1220.571,A -85,B 0,C 180,E1 15041.471,E2 15041.471} C_VEL
LIN {X 0,Y 447.461,Z 1215.219,A -85,B 0,C 180,E1 15043.834,E2 15043.834} C_VEL
LIN {X 0,Y 447.445,Z 1214.564,A -85,B 0,C 180,E1 15044.104,E2 15044.104} C_VEL
LIN {X 0,Y 449.671,Z 1198.176,A -85,B 0,C 180,E1 15049.381,E2 15049.381} C_VEL
LIN {X 0,Y 453.689,Z 1176.83,A -85,B 0,C 180,E1 15054.413,E2 15054.413} C_VEL
LIN {X 0,Y 460.007,Z 1148.688,A -85,B 0,C 180,E1 15059.377,E2 15059.377} C_VEL
LIN {X 0,Y 467.604,Z 1115.824,A -85,B 0,C 180,E1 15063.755,E2 15063.755} C_VEL
LIN {X 0,Y 476.232,Z 1076.935,A -85,B 0,C 180,E1 15067.626,E2 15067.626} C_VEL
LIN {X 0,Y 484.45,Z 1035.521,A -85,B 0,C 180,E1 15070.647,E2 15070.647} C_VEL
LIN {X 0,Y 491.444,Z 991.551,A -85,B 0,C 180,E1 15072.927,E2 15072.927} C_VEL
LIN {X 0,Y 494.83,Z 958.061,A -85,B 0,C 180,E1 15074.195,E2 15074.195} C_VEL
LIN {X 0,Y 480.983,Z 923.85,A -85,B 0,C 180,E1 15076.836,E2 15076.836} C_VEL
LIN {X 0,Y 460.498,Z 886.612,A -85,B 0,C 180,E1 15080.261,E2 15080.261} C_VEL
LIN {X 0,Y 445.97,Z 863.98,A -85,B 0,C 180,E1 15082.904,E2 15082.904} C_VEL
LIN {X 0,Y 444.421,Z 859.31,A -85,B 0,C 180,E1 15083.269,E2 15083.269} C_VEL
LIN {X 0,Y 444.527,Z 859.31,A -85,B 0,C 180,E1 15089.254,E2 15089.254} C_VEL
LIN {X 0,Y 444.839,Z 859.31,A -85,B 0,C 180,E1 15095.877,E2 15095.877} C_VEL
LIN {X 0,Y 445.103,Z 859.31,A -85,B 0,C 180,E1 15102.405,E2 15102.405} C_VEL
LIN {X 0,Y 445.306,Z 859.31,A -85,B 0,C 180,E1 15108.22,E2 15108.22} C_VEL
LIN {X 0,Y 445.755,Z 859.31,A -85,B 0,C 180,E1 15114.146,E2 15114.146} C_VEL
LIN {X 0,Y 446.113,Z 859.31,A -85,B 0,C 180,E1 15119.997,E2 15119.997} C_VEL
LIN {X 0,Y 445.766,Z 859.31,A -85,B 0,C 180,E1 15125.849,E2 15125.849} C_VEL
LIN {X 0,Y 445.367,Z 859.31,A -85,B 0,C 180,E1 15131.773,E2 15131.773} C_VEL
LIN {X 0,Y 445.064,Z 859.31,A -85,B 0,C 180,E1 15137.836,E2 15137.836} C_VEL
LIN {X 0,Y 444.794,Z 859.31,A -85,B 0,C 180,E1 15144.12,E2 15144.12} C_VEL
LIN {X 0,Y 444.512,Z 859.31,A -85,B 0,C 180,E1 15150.741,E2 15150.741} C_VEL
LIN {X 0,Y 444.4,Z 859.31,A -85,B 0,C 180,E1 15155.412,E2 15155.412} C_VEL
LIN {X 0,Y 444.299,Z 859.31,A -85,B 0,C 180,E1 15162.775,E2 15162.775} C_VEL
LIN {X 0,Y 446.783,Z 865.028,A -85,B 0,C 180,E1 15163.343,E2 15163.343} C_VEL
LIN {X 0,Y 468.403,Z 899.119,A -85,B 0,C 180,E1 15167.063,E2 15167.063} C_VEL
LIN {X 0,Y 489.396,Z 938.343,A -85,B 0,C 180,E1 15170.262,E2 15170.262} C_VEL
LIN {X 0,Y 496.897,Z 955.689,A -85,B 0,C 180,E1 15171.431,E2 15171.431} C_VEL
LIN {X 0,Y 492.733,Z 997.104,A -85,B 0,C 180,E1 15172.532,E2 15172.532} C_VEL
LIN {X 0,Y 486.648,Z 1036.249,A -85,B 0,C 180,E1 15174.28,E2 15174.28} C_VEL
LIN {X 0,Y 478.965,Z 1073.475,A -85,B 0,C 180,E1 15176.737,E2 15176.737} C_VEL
LIN {X 0,Y 470.849,Z 1106.688,A -85,B 0,C 180,E1 15179.813,E2 15179.813} C_VEL
LIN {X 0,Y 462.976,Z 1135.969,A -85,B 0,C 180,E1 15183.517,E2 15183.517} C_VEL
LIN {X 0,Y 456.228,Z 1160.842,A -85,B 0,C 180,E1 15187.803,E2 15187.803} C_VEL
LIN {X 0,Y 451.306,Z 1180.339,A -85,B 0,C 180,E1 15192.412,E2 15192.412} C_VEL
LIN {X 0,Y 448,Z 1196.01,A -85,B 0,C 180,E1 15197.796,E2 15197.796} C_VEL
LIN {X 0,Y 446.63,Z 1205.518,A -85,B 0,C 180,E1 15203.181,E2 15203.181} C_VEL
LIN {X 0,Y 446.237,Z 1209.417,A -85,B 0,C 180,E1 15208.054,E2 15208.054} C_VEL
LIN {X 0,Y 446.345,Z 1209.365,A -85,B 0,C 180,E1 15211.946,E2 15211.946} C_VEL
LIN {X 0,Y 446.661,Z 1205.401,A -85,B 0,C 180,E1 15216.819,E2 15216.819} C_VEL
LIN {X 0,Y 448.052,Z 1195.788,A -85,B 0,C 180,E1 15222.203,E2 15222.203} C_VEL
LIN {X 0,Y 451.327,Z 1180.012,A -85,B 0,C 180,E1 15227.588,E2 15227.588} C_VEL
LIN {X 0,Y 456.652,Z 1159.216,A -85,B 0,C 180,E1 15232.433,E2 15232.433} C_VEL
LIN {X 0,Y 463.581,Z 1133.786,A -85,B 0,C 180,E1 15236.708,E2 15236.708} C_VEL
LIN {X 0,Y 471.866,Z 1102.628,A -85,B 0,C 180,E1 15240.52,E2 15240.52} C_VEL
LIN {X 0,Y 479.996,Z 1068.642,A -85,B 0,C 180,E1 15243.536,E2 15243.536} C_VEL
LIN {X 0,Y 487.344,Z 1031.714,A -85,B 0,C 180,E1 15245.867,E2 15245.867} C_VEL
LIN {X 0,Y 493.294,Z 991.671,A -85,B 0,C 180,E1 15247.557,E2 15247.557} C_VEL
LIN {X 0,Y 496.376,Z 953.617,A -85,B 0,C 180,E1 15248.572,E2 15248.572} C_VEL
LIN {X 0,Y 475.792,Z 912.254,A -85,B 0,C 180,E1 15251.66,E2 15251.66} C_VEL
LIN {X 0,Y 454.318,Z 876.463,A -85,B 0,C 180,E1 15255.18,E2 15255.18} C_VEL
LIN {X 0,Y 446.027,Z 864.188,A -85,B 0,C 180,E1 15256.672,E2 15256.672} C_VEL
LIN {X 0,Y 444.303,Z 859.31,A -85,B 0,C 180,E1 15257.117,E2 15257.117} C_VEL
LIN {X 0,Y 444.31,Z 859.31,A -85,B 0,C 180,E1 15262.145,E2 15262.145} C_VEL
LIN {X 0,Y 444.482,Z 859.31,A -85,B 0,C 180,E1 15268.461,E2 15268.461} C_VEL
LIN {X 0,Y 444.642,Z 859.31,A -85,B 0,C 180,E1 15273.713,E2 15273.713} C_VEL
LIN {X 0,Y 444.872,Z 859.31,A -85,B 0,C 180,E1 15280.094,E2 15280.094} C_VEL
LIN {X 0,Y 445.157,Z 859.31,A -85,B 0,C 180,E1 15286.222,E2 15286.222} C_VEL
LIN {X 0,Y 445.622,Z 859.31,A -85,B 0,C 180,E1 15292.263,E2 15292.263} C_VEL
LIN {X 0,Y 445.972,Z 859.31,A -85,B 0,C 180,E1 15298.056,E2 15298.056} C_VEL
LIN {X 0,Y 445.87,Z 859.31,A -85,B 0,C 180,E1 15303.899,E2 15303.899} C_VEL
LIN {X 0,Y 445.474,Z 859.31,A -85,B 0,C 180,E1 15309.792,E2 15309.792} C_VEL
LIN {X 0,Y 445.157,Z 859.31,A -85,B 0,C 180,E1 15315.801,E2 15315.801} C_VEL
LIN {X 0,Y 444.919,Z 859.31,A -85,B 0,C 180,E1 15321.998,E2 15321.998} C_VEL
LIN {X 0,Y 444.615,Z 859.31,A -85,B 0,C 180,E1 15328.493,E2 15328.493} C_VEL
LIN {X 0,Y 444.406,Z 859.31,A -85,B 0,C 180,E1 15335.418,E2 15335.418} C_VEL
LIN {X 0,Y 444.457,Z 859.732,A -85,B 0,C 180,E1 15336.782,E2 15336.782} C_VEL
LIN {X 0,Y 446.801,Z 864.966,A -85,B 0,C 180,E1 15337.277,E2 15337.277} C_VEL
LIN {X 0,Y 468.062,Z 899.737,A -85,B 0,C 180,E1 15341.056,E2 15341.056} C_VEL
LIN {X 0,Y 487.036,Z 937.387,A -85,B 0,C 180,E1 15344.255,E2 15344.255} C_VEL
LIN {X 0,Y 495.219,Z 960.393,A -85,B 0,C 180,E1 15345.948,E2 15345.948} C_VEL
LIN {X 0,Y 489.436,Z 1004.601,A -85,B 0,C 180,E1 15347.669,E2 15347.669} C_VEL
LIN {X 0,Y 482.369,Z 1046.057,A -85,B 0,C 180,E1 15350.043,E2 15350.043} C_VEL
LIN {X 0,Y 474.451,Z 1084.783,A -85,B 0,C 180,E1 15353.079,E2 15353.079} C_VEL
LIN {X 0,Y 466.616,Z 1119.884,A -85,B 0,C 180,E1 15356.741,E2 15356.741} C_VEL
LIN {X 0,Y 459.46,Z 1150.959,A -85,B 0,C 180,E1 15360.981,E2 15360.981} C_VEL
LIN {X 0,Y 453.261,Z 1179.239,A -85,B 0,C 180,E1 15366.087,E2 15366.087} C_VEL
LIN {X 0,Y 449.197,Z 1201.197,A -85,B 0,C 180,E1 15371.452,E2 15371.452} C_VEL
LIN {X 0,Y 447.19,Z 1216.702,A -85,B 0,C 180,E1 15376.778,E2 15376.778} C_VEL
LIN {X 0,Y 446.472,Z 1225.548,A -85,B 0,C 180,E1 15381.215,E2 15381.215} C_VEL
LIN {X 0,Y 446.148,Z 1231.146,A -85,B 0,C 180,E1 15386.105,E2 15386.105} C_VEL
LIN {X 0,Y 446.258,Z 1232.552,A -85,B 0,C 180,E1 15390,E2 15390} C_VEL
LIN {X 0,Y 446.196,Z 1231.151,A -85,B 0,C 180,E1 15393.894,E2 15393.894} C_VEL
LIN {X 0,Y 446.428,Z 1225.556,A -85,B 0,C 180,E1 15398.786,E2 15398.786} C_VEL
LIN {X 0,Y 447.445,Z 1214.564,A -85,B 0,C 180,E1 15404.104,E2 15404.104} C_VEL
LIN {X 0,Y 444.206,Z 1209.081,A -85,B 0,C 180,E1 15406.204,E2 15406.204} C_VEL
LIN {X 0,Y 441.209,Z 1202.872,A -85,B 0,C 180,E1 15408.302,E2 15408.302} C_VEL
LIN {X 0,Y 445.262,Z 1181.411,A -85,B 0,C 180,E1 15413.799,E2 15413.799} C_VEL
LIN {X 0,Y 451.067,Z 1155.367,A -85,B 0,C 180,E1 15418.759,E2 15418.759} C_VEL
LIN {X 0,Y 458.344,Z 1125.712,A -85,B 0,C 180,E1 15423.058,E2 15423.058} C_VEL
LIN {X 0,Y 466.834,Z 1089.552,A -85,B 0,C 180,E1 15427.046,E2 15427.046} C_VEL
LIN {X 0,Y 475.18,Z 1050.786,A -85,B 0,C 180,E1 15430.232,E2 15430.232} C_VEL
LIN {X 0,Y 482.982,Z 1007.264,A -85,B 0,C 180,E1 15432.816,E2 15432.816} C_VEL
LIN {X 0,Y 488.834,Z 961.104,A -85,B 0,C 180,E1 15434.694,E2 15434.694} C_VEL
LIN {X 0,Y 475.063,Z 926.733,A -85,B 0,C 180,E1 15437.45,E2 15437.45} C_VEL
LIN {X 0,Y 454.125,Z 888.629,A -85,B 0,C 180,E1 15441.086,E2 15441.086} C_VEL
LIN {X 0,Y 438.411,Z 864.45,A -85,B 0,C 180,E1 15444.075,E2 15444.075} C_VEL
LIN {X 0,Y 436.514,Z 859.31,A -85,B 0,C 180,E1 15444.64,E2 15444.64} C_VEL
LIN {X 0,Y 436.645,Z 859.31,A -85,B 0,C 180,E1 15450.938,E2 15450.938} C_VEL
LIN {X 0,Y 437.011,Z 859.31,A -85,B 0,C 180,E1 15457.582,E2 15457.582} C_VEL
LIN {X 0,Y 437.192,Z 859.31,A -85,B 0,C 180,E1 15463.904,E2 15463.904} C_VEL
LIN {X 0,Y 437.54,Z 859.31,A -85,B 0,C 180,E1 15470.028,E2 15470.028} C_VEL
LIN {X 0,Y 437.979,Z 859.31,A -85,B 0,C 180,E1 15476.031,E2 15476.031} C_VEL
LIN {X 0,Y 438.154,Z 859.31,A -85,B 0,C 180,E1 15481.979,E2 15481.979} C_VEL
LIN {X 0,Y 437.656,Z 859.31,A -85,B 0,C 180,E1 15487.956,E2 15487.956} C_VEL
LIN {X 0,Y 437.326,Z 859.31,A -85,B 0,C 180,E1 15494.03,E2 15494.03} C_VEL
LIN {X 0,Y 437.034,Z 859.31,A -85,B 0,C 180,E1 15500.586,E2 15500.586} C_VEL
LIN {X 0,Y 436.693,Z 859.31,A -85,B 0,C 180,E1 15506.803,E2 15506.803} C_VEL
LIN {X 0,Y 436.477,Z 859.31,A -85,B 0,C 180,E1 15513.729,E2 15513.729} C_VEL
LIN {X 0,Y 436.312,Z 859.31,A -85,B 0,C 180,E1 15520.178,E2 15520.178} C_VEL
LIN {X 0,Y 436.384,Z 860.08,A -85,B 0,C 180,E1 15521.58,E2 15521.58} C_VEL
LIN {X 0,Y 439.281,Z 865.428,A -85,B 0,C 180,E1 15522.18,E2 15522.18} C_VEL
LIN {X 0,Y 461.903,Z 901.01,A -85,B 0,C 180,E1 15526.259,E2 15526.259} C_VEL
LIN {X 0,Y 482.443,Z 938.937,A -85,B 0,C 180,E1 15529.503,E2 15529.503} C_VEL
LIN {X 0,Y 490.836,Z 957.605,A -85,B 0,C 180,E1 15530.857,E2 15530.857} C_VEL
LIN {X 0,Y 486.551,Z 998.21,A -85,B 0,C 180,E1 15531.971,E2 15531.971} C_VEL
LIN {X 0,Y 480.57,Z 1035.568,A -85,B 0,C 180,E1 15533.655,E2 15533.655} C_VEL
LIN {X 0,Y 472.925,Z 1071.786,A -85,B 0,C 180,E1 15536.035,E2 15536.035} C_VEL
LIN {X 0,Y 464.315,Z 1106.034,A -85,B 0,C 180,E1 15539.206,E2 15539.206} C_VEL
LIN {X 0,Y 455.864,Z 1136.276,A -85,B 0,C 180,E1 15543.071,E2 15543.071} C_VEL
LIN {X 0,Y 448.811,Z 1161.106,A -85,B 0,C 180,E1 15547.416,E2 15547.416} C_VEL
LIN {X 0,Y 443.664,Z 1180.573,A -85,B 0,C 180,E1 15552.098,E2 15552.098} C_VEL
LIN {X 0,Y 440.418,Z 1195.127,A -85,B 0,C 180,E1 15557.077,E2 15557.077} C_VEL
LIN {X 0,Y 438.869,Z 1204.426,A -85,B 0,C 180,E1 15562.062,E2 15562.062} C_VEL
LIN {X 0,Y 438.453,Z 1208.59,A -85,B 0,C 180,E1 15566.037,E2 15566.037} C_VEL
LIN {X 0,Y 438.379,Z 1209.944,A -85,B 0,C 180,E1 15570,E2 15570} C_VEL
LIN {X 0,Y 438.455,Z 1208.507,A -85,B 0,C 180,E1 15573.964,E2 15573.964} C_VEL
LIN {X 0,Y 439.126,Z 1202.799,A -85,B 0,C 180,E1 15578.933,E2 15578.933} C_VEL
LIN {X 0,Y 441.267,Z 1191.057,A -85,B 0,C 180,E1 15584.416,E2 15584.416} C_VEL
LIN {X 0,Y 445.607,Z 1172.736,A -85,B 0,C 180,E1 15589.88,E2 15589.88} C_VEL
LIN {X 0,Y 451.71,Z 1150.621,A -85,B 0,C 180,E1 15594.496,E2 15594.496} C_VEL
LIN {X 0,Y 459.334,Z 1123.839,A -85,B 0,C 180,E1 15598.577,E2 15598.577} C_VEL
LIN {X 0,Y 467.981,Z 1091.639,A -85,B 0,C 180,E1 15602.157,E2 15602.157} C_VEL
LIN {X 0,Y 476.174,Z 1056.909,A -85,B 0,C 180,E1 15604.946,E2 15604.946} C_VEL
LIN {X 0,Y 483.27,Z 1019.631,A -85,B 0,C 180,E1 15607.054,E2 15607.054} C_VEL
LIN {X 0,Y 488.793,Z 979.229,A -85,B 0,C 180,E1 15608.538,E2 15608.538} C_VEL
LIN {X 0,Y 490.175,Z 956.01,A -85,B 0,C 180,E1 15609.152,E2 15609.152} C_VEL
LIN {X 0,Y 470.5,Z 916.251,A -85,B 0,C 180,E1 15612.226,E2 15612.226} C_VEL
LIN {X 0,Y 449.949,Z 881.764,A -85,B 0,C 180,E1 15615.695,E2 15615.695} C_VEL
LIN {X 0,Y 438.435,Z 864.609,A -85,B 0,C 180,E1 15617.85,E2 15617.85} C_VEL
LIN {X 0,Y 436.335,Z 859.31,A -85,B 0,C 180,E1 15618.477,E2 15618.477} C_VEL
LIN {X 0,Y 436.399,Z 859.31,A -85,B 0,C 180,E1 15623.837,E2 15623.837} C_VEL
LIN {X 0,Y 436.583,Z 859.31,A -85,B 0,C 180,E1 15630.193,E2 15630.193} C_VEL
LIN {X 0,Y 436.789,Z 859.31,A -85,B 0,C 180,E1 15635.409,E2 15635.409} C_VEL
LIN {X 0,Y 436.978,Z 859.31,A -85,B 0,C 180,E1 15641.823,E2 15641.823} C_VEL
LIN {X 0,Y 437.346,Z 859.31,A -85,B 0,C 180,E1 15648.008,E2 15648.008} C_VEL
LIN {X 0,Y 437.849,Z 859.31,A -85,B 0,C 180,E1 15654.045,E2 15654.045} C_VEL
LIN {X 0,Y 438.231,Z 859.31,A -85,B 0,C 180,E1 15660.003,E2 15660.003} C_VEL
LIN {X 0,Y 437.838,Z 859.31,A -85,B 0,C 180,E1 15665.961,E2 15665.961} C_VEL
LIN {X 0,Y 437.392,Z 859.31,A -85,B 0,C 180,E1 15671.997,E2 15671.997} C_VEL
LIN {X 0,Y 437.133,Z 859.31,A -85,B 0,C 180,E1 15678.176,E2 15678.176} C_VEL
LIN {X 0,Y 436.835,Z 859.31,A -85,B 0,C 180,E1 15684.594,E2 15684.594} C_VEL
LIN {X 0,Y 436.609,Z 859.31,A -85,B 0,C 180,E1 15691.366,E2 15691.366} C_VEL
LIN {X 0,Y 436.536,Z 859.31,A -85,B 0,C 180,E1 15695.486,E2 15695.486} C_VEL
LIN {X 0,Y 438.873,Z 864.902,A -85,B 0,C 180,E1 15696.04,E2 15696.04} C_VEL
LIN {X 0,Y 460.425,Z 899.428,A -85,B 0,C 180,E1 15700.061,E2 15700.061} C_VEL
LIN {X 0,Y 479.857,Z 937.483,A -85,B 0,C 180,E1 15703.461,E2 15703.461} C_VEL
LIN {X 0,Y 489.056,Z 962.27,A -85,B 0,C 180,E1 15705.398,E2 15705.398} C_VEL
LIN {X 0,Y 482.89,Z 1007.357,A -85,B 0,C 180,E1 15707.195,E2 15707.195} C_VEL
LIN {X 0,Y 475.242,Z 1050.401,A -85,B 0,C 180,E1 15709.753,E2 15709.753} C_VEL
LIN {X 0,Y 466.628,Z 1090.582,A -85,B 0,C 180,E1 15713.063,E2 15713.063} C_VEL
LIN {X 0,Y 457.717,Z 1128.069,A -85,B 0,C 180,E1 15717.241,E2 15717.241} C_VEL
LIN {X 0,Y 449.939,Z 1160.294,A -85,B 0,C 180,E1 15722.07,E2 15722.07} C_VEL
LIN {X 0,Y 444.285,Z 1186.859,A -85,B 0,C 180,E1 15727.433,E2 15727.433} C_VEL
LIN {X 0,Y 440.603,Z 1206.991,A -85,B 0,C 180,E1 15733.002,E2 15733.002} C_VEL
LIN {X 0,Y 439.028,Z 1219.841,A -85,B 0,C 180,E1 15738.048,E2 15738.048} C_VEL
LIN {X 0,Y 438.471,Z 1228.08,A -85,B 0,C 180,E1 15743.053,E2 15743.053} C_VEL
LIN {X 0,Y 438.364,Z 1231.993,A -85,B 0,C 180,E1 15748.019,E2 15748.019} C_VEL
LIN {X 0,Y 438.327,Z 1231.993,A -85,B 0,C 180,E1 15751.981,E2 15751.981} C_VEL
LIN {X 0,Y 438.459,Z 1228.088,A -85,B 0,C 180,E1 15756.947,E2 15756.947} C_VEL
LIN {X 0,Y 439.148,Z 1218.838,A -85,B 0,C 180,E1 15762.454,E2 15762.454} C_VEL
LIN {X 0,Y 441.059,Z 1203.797,A -85,B 0,C 180,E1 15768.011,E2 15768.011} C_VEL
LIN {X 0,Y 441.209,Z 1202.872,A -85,B 0,C 180,E1 15768.302,E2 15768.302} C_VEL
LIN {X 0,Y 438.588,Z 1196.147,A -85,B 0,C 180,E1 15770.382,E2 15770.382} C_VEL
LIN {X 0,Y 436.261,Z 1188.736,A -85,B 0,C 180,E1 15772.447,E2 15772.447} C_VEL
LIN {X 0,Y 441.592,Z 1165.092,A -85,B 0,C 180,E1 15777.485,E2 15777.485} C_VEL
LIN {X 0,Y 448.766,Z 1135.73,A -85,B 0,C 180,E1 15782.233,E2 15782.233} C_VEL
LIN {X 0,Y 457.193,Z 1102.436,A -85,B 0,C 180,E1 15786.305,E2 15786.305} C_VEL
LIN {X 0,Y 465.92,Z 1064.433,A -85,B 0,C 180,E1 15789.813,E2 15789.813} C_VEL
LIN {X 0,Y 474.518,Z 1021.385,A -85,B 0,C 180,E1 15792.688,E2 15792.688} C_VEL
LIN {X 0,Y 481.519,Z 976.753,A -85,B 0,C 180,E1 15794.738,E2 15794.738} C_VEL
LIN {X 0,Y 482.491,Z 962.811,A -85,B 0,C 180,E1 15795.293,E2 15795.293} C_VEL
LIN {X 0,Y 468.217,Z 927.63,A -85,B 0,C 180,E1 15798.253,E2 15798.253} C_VEL
LIN {X 0,Y 448.475,Z 892.092,A -85,B 0,C 180,E1 15801.808,E2 15801.808} C_VEL
LIN {X 0,Y 430.975,Z 864.957,A -85,B 0,C 180,E1 15805.3,E2 15805.3} C_VEL
LIN {X 0,Y 428.59,Z 859.31,A -85,B 0,C 180,E1 15806.01,E2 15806.01} C_VEL
LIN {X 0,Y 428.767,Z 859.31,A -85,B 0,C 180,E1 15812.655,E2 15812.655} C_VEL
LIN {X 0,Y 429.143,Z 859.31,A -85,B 0,C 180,E1 15819.326,E2 15819.326} C_VEL
LIN {X 0,Y 429.352,Z 859.31,A -85,B 0,C 180,E1 15825.698,E2 15825.698} C_VEL
LIN {X 0,Y 429.734,Z 859.31,A -85,B 0,C 180,E1 15831.891,E2 15831.891} C_VEL
LIN {X 0,Y 430.161,Z 859.31,A -85,B 0,C 180,E1 15837.979,E2 15837.979} C_VEL
LIN {X 0,Y 430.053,Z 859.31,A -85,B 0,C 180,E1 15844.037,E2 15844.037} C_VEL
LIN {X 0,Y 429.627,Z 859.31,A -85,B 0,C 180,E1 15850.152,E2 15850.152} C_VEL
LIN {X 0,Y 429.272,Z 859.31,A -85,B 0,C 180,E1 15856.396,E2 15856.396} C_VEL
LIN {X 0,Y 428.923,Z 859.31,A -85,B 0,C 180,E1 15863.289,E2 15863.289} C_VEL
LIN {X 0,Y 428.692,Z 859.31,A -85,B 0,C 180,E1 15869.648,E2 15869.648} C_VEL
LIN {X 0,Y 428.447,Z 859.31,A -85,B 0,C 180,E1 15876.944,E2 15876.944} C_VEL
LIN {X 0,Y 428.412,Z 859.461,A -85,B 0,C 180,E1 15880.2,E2 15880.2} C_VEL
LIN {X 0,Y 430.783,Z 864.945,A -85,B 0,C 180,E1 15880.753,E2 15880.753} C_VEL
LIN {X 0,Y 448.789,Z 892.004,A -85,B 0,C 180,E1 15884.245,E2 15884.245} C_VEL
LIN {X 0,Y 470.285,Z 929.285,A -85,B 0,C 180,E1 15887.889,E2 15887.889} C_VEL
LIN {X 0,Y 484.793,Z 960.6,A -85,B 0,C 180,E1 15890.296,E2 15890.296} C_VEL
LIN {X 0,Y 480.194,Z 1000.732,A -85,B 0,C 180,E1 15891.448,E2 15891.448} C_VEL
LIN {X 0,Y 473.857,Z 1038.244,A -85,B 0,C 180,E1 15893.205,E2 15893.205} C_VEL
LIN {X 0,Y 466.069,Z 1073.634,A -85,B 0,C 180,E1 15895.605,E2 15895.605} C_VEL
LIN {X 0,Y 457.501,Z 1106.409,A -85,B 0,C 180,E1 15898.696,E2 15898.696} C_VEL
LIN {X 0,Y 449.232,Z 1135.029,A -85,B 0,C 180,E1 15902.368,E2 15902.368} C_VEL
LIN {X 0,Y 441.78,Z 1160.208,A -85,B 0,C 180,E1 15906.769,E2 15906.769} C_VEL
LIN {X 0,Y 436.072,Z 1180.805,A -85,B 0,C 180,E1 15911.776,E2 15911.776} C_VEL
LIN {X 0,Y 432.648,Z 1195.346,A -85,B 0,C 180,E1 15916.841,E2 15916.841} C_VEL
LIN {X 0,Y 431.001,Z 1204.635,A -85,B 0,C 180,E1 15921.916,E2 15921.916} C_VEL
LIN {X 0,Y 430.556,Z 1208.794,A -85,B 0,C 180,E1 15925.964,E2 15925.964} C_VEL
LIN {X 0,Y 430.481,Z 1210.146,A -85,B 0,C 180,E1 15930,E2 15930} C_VEL
LIN {X 0,Y 430.559,Z 1208.712,A -85,B 0,C 180,E1 15934.036,E2 15934.036} C_VEL
LIN {X 0,Y 431.282,Z 1203.008,A -85,B 0,C 180,E1 15939.097,E2 15939.097} C_VEL
LIN {X 0,Y 433.563,Z 1191.278,A -85,B 0,C 180,E1 15944.678,E2 15944.678} C_VEL
LIN {X 0,Y 438.095,Z 1172.992,A -85,B 0,C 180,E1 15950.236,E2 15950.236} C_VEL
LIN {X 0,Y 444.687,Z 1150.156,A -85,B 0,C 180,E1 15955.054,E2 15955.054} C_VEL
LIN {X 0,Y 452.893,Z 1122.202,A -85,B 0,C 180,E1 15959.315,E2 15959.315} C_VEL
LIN {X 0,Y 461.729,Z 1090.436,A -85,B 0,C 180,E1 15962.833,E2 15962.833} C_VEL
LIN {X 0,Y 470.13,Z 1055.9,A -85,B 0,C 180,E1 15965.6,E2 15965.6} C_VEL
LIN {X 0,Y 477.44,Z 1018.098,A -85,B 0,C 180,E1 15967.731,E2 15967.731} C_VEL
LIN {X 0,Y 482.904,Z 978.95,A -85,B 0,C 180,E1 15969.168,E2 15969.168} C_VEL
LIN {X 0,Y 484.292,Z 959.041,A -85,B 0,C 180,E1 15969.695,E2 15969.695} C_VEL
LIN {X 0,Y 465.077,Z 919.803,A -85,B 0,C 180,E1 15972.837,E2 15972.837} C_VEL
LIN {X 0,Y 443.55,Z 883.524,A -85,B 0,C 180,E1 15976.61,E2 15976.61} C_VEL
LIN {X 0,Y 430.551,Z 864.719,A -85,B 0,C 180,E1 15979.167,E2 15979.167} C_VEL
LIN {X 0,Y 428.428,Z 859.31,A -85,B 0,C 180,E1 15979.702,E2 15979.702} C_VEL
LIN {X 0,Y 428.483,Z 859.31,A -85,B 0,C 180,E1 15985.554,E2 15985.554} C_VEL
LIN {X 0,Y 428.702,Z 859.31,A -85,B 0,C 180,E1 15992.087,E2 15992.087} C_VEL
LIN {X 0,Y 428.923,Z 859.31,A -85,B 0,C 180,E1 15997.142,E2 15997.142} C_VEL
LIN {X 0,Y 429.101,Z 859.31,A -85,B 0,C 180,E1 16003.598,E2 16003.598} C_VEL
LIN {X 0,Y 429.64,Z 859.31,A -85,B 0,C 180,E1 16009.849,E2 16009.849} C_VEL
LIN {X 0,Y 430.069,Z 859.31,A -85,B 0,C 180,E1 16015.963,E2 16015.963} C_VEL
LIN {X 0,Y 430.248,Z 859.31,A -85,B 0,C 180,E1 16022.021,E2 16022.021} C_VEL
LIN {X 0,Y 429.719,Z 859.31,A -85,B 0,C 180,E1 16028.109,E2 16028.109} C_VEL
LIN {X 0,Y 429.392,Z 859.31,A -85,B 0,C 180,E1 16034.3,E2 16034.3} C_VEL
LIN {X 0,Y 429.144,Z 859.31,A -85,B 0,C 180,E1 16040.674,E2 16040.674} C_VEL
LIN {X 0,Y 428.736,Z 859.31,A -85,B 0,C 180,E1 16047.348,E2 16047.348} C_VEL
LIN {X 0,Y 428.605,Z 859.31,A -85,B 0,C 180,E1 16054.153,E2 16054.153} C_VEL
LIN {X 0,Y 430.852,Z 864.824,A -85,B 0,C 180,E1 16054.711,E2 16054.711} C_VEL
LIN {X 0,Y 448.295,Z 891.911,A -85,B 0,C 180,E1 16058.188,E2 16058.188} C_VEL
LIN {X 0,Y 468.045,Z 927.559,A -85,B 0,C 180,E1 16061.745,E2 16061.745} C_VEL
LIN {X 0,Y 482.114,Z 961.932,A -85,B 0,C 180,E1 16064.641,E2 16064.641} C_VEL
LIN {X 0,Y 482.387,Z 968.01,A -85,B 0,C 180,E1 16064.958,E2 16064.958} C_VEL
LIN {X 0,Y 476.538,Z 1009.111,A -85,B 0,C 180,E1 16066.672,E2 16066.672} C_VEL
LIN {X 0,Y 468.639,Z 1051.802,A -85,B 0,C 180,E1 16069.258,E2 16069.258} C_VEL
LIN {X 0,Y 459.698,Z 1091.903,A -85,B 0,C 180,E1 16072.627,E2 16072.627} C_VEL
LIN {X 0,Y 451.009,Z 1127.217,A -85,B 0,C 180,E1 16076.621,E2 16076.621} C_VEL
LIN {X 0,Y 442.639,Z 1160.351,A -85,B 0,C 180,E1 16081.642,E2 16081.642} C_VEL
LIN {X 0,Y 436.712,Z 1186.581,A -85,B 0,C 180,E1 16087.019,E2 16087.019} C_VEL
LIN {X 0,Y 432.841,Z 1206.743,A -85,B 0,C 180,E1 16092.688,E2 16092.688} C_VEL
LIN {X 0,Y 431.099,Z 1220.635,A -85,B 0,C 180,E1 16098.339,E2 16098.339} C_VEL
LIN {X 0,Y 430.516,Z 1229.01,A -85,B 0,C 180,E1 16103.939,E2 16103.939} C_VEL
LIN {X 0,Y 430.458,Z 1231.791,A -85,B 0,C 180,E1 16107.982,E2 16107.982} C_VEL
LIN {X 0,Y 430.423,Z 1231.791,A -85,B 0,C 180,E1 16112.017,E2 16112.017} C_VEL
LIN {X 0,Y 430.55,Z 1227.878,A -85,B 0,C 180,E1 16117.075,E2 16117.075} C_VEL
LIN {X 0,Y 431.323,Z 1218.617,A -85,B 0,C 180,E1 16122.684,E2 16122.684} C_VEL
LIN {X 0,Y 433.355,Z 1203.395,A -85,B 0,C 180,E1 16128.394,E2 16128.394} C_VEL
LIN {X 0,Y 436.261,Z 1188.736,A -85,B 0,C 180,E1 16132.447,E2 16132.447} C_VEL
LIN {X 0,Y 434.156,Z 1180.87,A -85,B 0,C 180,E1 16134.491,E2 16134.491} C_VEL
LIN {X 0,Y 432.452,Z 1172.346,A -85,B 0,C 180,E1 16136.505,E2 16136.505} C_VEL
LIN {X 0,Y 439.489,Z 1144.787,A -85,B 0,C 180,E1 16141.395,E2 16141.395} C_VEL
LIN {X 0,Y 447.704,Z 1112.965,A -85,B 0,C 180,E1 16145.695,E2 16145.695} C_VEL
LIN {X 0,Y 456.994,Z 1075.679,A -85,B 0,C 180,E1 16149.471,E2 16149.471} C_VEL
LIN {X 0,Y 465.775,Z 1035.639,A -85,B 0,C 180,E1 16152.458,E2 16152.458} C_VEL
LIN {X 0,Y 473.43,Z 992.155,A -85,B 0,C 180,E1 16154.76,E2 16154.76} C_VEL
LIN {X 0,Y 476.362,Z 965.581,A -85,B 0,C 180,E1 16155.838,E2 16155.838} C_VEL
LIN {X 0,Y 462.719,Z 931.212,A -85,B 0,C 180,E1 16158.839,E2 16158.839} C_VEL
LIN {X 0,Y 442.782,Z 894.965,A -85,B 0,C 180,E1 16162.58,E2 16162.58} C_VEL
LIN {X 0,Y 423.579,Z 865.404,A -85,B 0,C 180,E1 16166.597,E2 16166.597} C_VEL
LIN {X 0,Y 420.849,Z 860.952,A -85,B 0,C 180,E1 16167.237,E2 16167.237} C_VEL
LIN {X 0,Y 420.678,Z 859.31,A -85,B 0,C 180,E1 16167.445,E2 16167.445} C_VEL
LIN {X 0,Y 420.915,Z 859.31,A -85,B 0,C 180,E1 16174.41,E2 16174.41} C_VEL
LIN {X 0,Y 421.227,Z 859.31,A -85,B 0,C 180,E1 16181.112,E2 16181.112} C_VEL
LIN {X 0,Y 421.508,Z 859.31,A -85,B 0,C 180,E1 16187.544,E2 16187.544} C_VEL
LIN {X 0,Y 422.008,Z 859.31,A -85,B 0,C 180,E1 16193.815,E2 16193.815} C_VEL
LIN {X 0,Y 422.434,Z 859.31,A -85,B 0,C 180,E1 16199.997,E2 16199.997} C_VEL
LIN {X 0,Y 422.014,Z 859.31,A -85,B 0,C 180,E1 16206.179,E2 16206.179} C_VEL
LIN {X 0,Y 421.557,Z 859.31,A -85,B 0,C 180,E1 16212.449,E2 16212.449} C_VEL
LIN {X 0,Y 421.215,Z 859.31,A -85,B 0,C 180,E1 16218.883,E2 16218.883} C_VEL
LIN {X 0,Y 420.844,Z 859.31,A -85,B 0,C 180,E1 16225.823,E2 16225.823} C_VEL
LIN {X 0,Y 420.587,Z 859.31,A -85,B 0,C 180,E1 16232.699,E2 16232.699} C_VEL
LIN {X 0,Y 420.544,Z 859.31,A -85,B 0,C 180,E1 16238.728,E2 16238.728} C_VEL
LIN {X 0,Y 422.834,Z 864.9,A -85,B 0,C 180,E1 16239.331,E2 16239.331} C_VEL
LIN {X 0,Y 440.765,Z 891.307,A -85,B 0,C 180,E1 16243.018,E2 16243.018} C_VEL
LIN {X 0,Y 461.266,Z 926.143,A -85,B 0,C 180,E1 16246.686,E2 16246.686} C_VEL
LIN {X 0,Y 478.7,Z 962.704,A -85,B 0,C 180,E1 16249.685,E2 16249.685} C_VEL
LIN {X 0,Y 473.873,Z 1003.242,A -85,B 0,C 180,E1 16250.91,E2 16250.91} C_VEL
LIN {X 0,Y 467.224,Z 1040.661,A -85,B 0,C 180,E1 16252.728,E2 16252.728} C_VEL
LIN {X 0,Y 459.197,Z 1075.492,A -85,B 0,C 180,E1 16255.16,E2 16255.16} C_VEL
LIN {X 0,Y 450.426,Z 1107.808,A -85,B 0,C 180,E1 16258.289,E2 16258.289} C_VEL
LIN {X 0,Y 441.705,Z 1136.883,A -85,B 0,C 180,E1 16262.134,E2 16262.134} C_VEL
LIN {X 0,Y 434.065,Z 1161.626,A -85,B 0,C 180,E1 16266.604,E2 16266.604} C_VEL
LIN {X 0,Y 428.484,Z 1181.037,A -85,B 0,C 180,E1 16271.442,E2 16271.442} C_VEL
LIN {X 0,Y 424.888,Z 1195.562,A -85,B 0,C 180,E1 16276.597,E2 16276.597} C_VEL
LIN {X 0,Y 423.155,Z 1204.842,A -85,B 0,C 180,E1 16281.765,E2 16281.765} C_VEL
LIN {X 0,Y 422.676,Z 1208.997,A -85,B 0,C 180,E1 16285.889,E2 16285.889} C_VEL
LIN {X 0,Y 422.608,Z 1210.347,A -85,B 0,C 180,E1 16290,E2 16290} C_VEL
LIN {X 0,Y 422.68,Z 1208.916,A -85,B 0,C 180,E1 16294.112,E2 16294.112} C_VEL
LIN {X 0,Y 423.427,Z 1203.217,A -85,B 0,C 180,E1 16299.267,E2 16299.267} C_VEL
LIN {X 0,Y 425.844,Z 1191.5,A -85,B 0,C 180,E1 16304.95,E2 16304.95} C_VEL
LIN {X 0,Y 430.625,Z 1173.245,A -85,B 0,C 180,E1 16310.603,E2 16310.603} C_VEL
LIN {X 0,Y 437.665,Z 1149.766,A -85,B 0,C 180,E1 16315.617,E2 16315.617} C_VEL
LIN {X 0,Y 445.854,Z 1123.003,A -85,B 0,C 180,E1 16319.757,E2 16319.757} C_VEL
LIN {X 0,Y 455.093,Z 1090.882,A -85,B 0,C 180,E1 16323.375,E2 16323.375} C_VEL
LIN {X 0,Y 463.696,Z 1056.771,A -85,B 0,C 180,E1 16326.15,E2 16326.15} C_VEL
LIN {X 0,Y 471.27,Z 1019.043,A -85,B 0,C 180,E1 16328.313,E2 16328.313} C_VEL
LIN {X 0,Y 477.076,Z 978.948,A -85,B 0,C 180,E1 16329.803,E2 16329.803} C_VEL
LIN {X 0,Y 478.2,Z 961.584,A -85,B 0,C 180,E1 16330.295,E2 16330.295} C_VEL
LIN {X 0,Y 459.732,Z 923.456,A -85,B 0,C 180,E1 16333.455,E2 16333.455} C_VEL
LIN {X 0,Y 439.135,Z 888.729,A -85,B 0,C 180,E1 16337.173,E2 16337.173} C_VEL
LIN {X 0,Y 423.051,Z 865.093,A -85,B 0,C 180,E1 16340.489,E2 16340.489} C_VEL
LIN {X 0,Y 420.592,Z 859.767,A -85,B 0,C 180,E1 16341.091,E2 16341.091} C_VEL
LIN {X 0,Y 420.597,Z 859.31,A -85,B 0,C 180,E1 16347.302,E2 16347.302} C_VEL
LIN {X 0,Y 420.86,Z 859.31,A -85,B 0,C 180,E1 16354.412,E2 16354.412} C_VEL
LIN {X 0,Y 421.093,Z 859.31,A -85,B 0,C 180,E1 16361.111,E2 16361.111} C_VEL
LIN {X 0,Y 421.472,Z 859.31,A -85,B 0,C 180,E1 16367.549,E2 16367.549} C_VEL
LIN {X 0,Y 422.028,Z 859.31,A -85,B 0,C 180,E1 16373.821,E2 16373.821} C_VEL
LIN {X 0,Y 422.438,Z 859.31,A -85,B 0,C 180,E1 16380.003,E2 16380.003} C_VEL
LIN {X 0,Y 422.012,Z 859.31,A -85,B 0,C 180,E1 16386.185,E2 16386.185} C_VEL
LIN {X 0,Y 421.533,Z 859.31,A -85,B 0,C 180,E1 16392.455,E2 16392.455} C_VEL
LIN {X 0,Y 421.234,Z 859.31,A -85,B 0,C 180,E1 16398.888,E2 16398.888} C_VEL
LIN {X 0,Y 420.894,Z 859.31,A -85,B 0,C 180,E1 16405.592,E2 16405.592} C_VEL
LIN {X 0,Y 420.709,Z 859.31,A -85,B 0,C 180,E1 16412.695,E2 16412.695} C_VEL
LIN {X 0,Y 422.926,Z 864.821,A -85,B 0,C 180,E1 16413.302,E2 16413.302} C_VEL
LIN {X 0,Y 430.144,Z 875.435,A -85,B 0,C 180,E1 16414.89,E2 16414.89} C_VEL
LIN {X 0,Y 450.349,Z 908.094,A -85,B 0,C 180,E1 16418.892,E2 16418.892} C_VEL
LIN {X 0,Y 468.503,Z 944.38,A -85,B 0,C 180,E1 16422.362,E2 16422.362} C_VEL
LIN {X 0,Y 476.628,Z 967.451,A -85,B 0,C 180,E1 16424.3,E2 16424.3} C_VEL
LIN {X 0,Y 470.452,Z 1009.51,A -85,B 0,C 180,E1 16426.061,E2 16426.061} C_VEL
LIN {X 0,Y 462.524,Z 1051.133,A -85,B 0,C 180,E1 16428.595,E2 16428.595} C_VEL
LIN {X 0,Y 453.388,Z 1090.673,A -85,B 0,C 180,E1 16431.922,E2 16431.922} C_VEL
LIN {X 0,Y 444.193,Z 1126.826,A -85,B 0,C 180,E1 16436.04,E2 16436.04} C_VEL
LIN {X 0,Y 435.831,Z 1158.56,A -85,B 0,C 180,E1 16440.872,E2 16440.872} C_VEL
LIN {X 0,Y 429.383,Z 1185.187,A -85,B 0,C 180,E1 16446.331,E2 16446.331} C_VEL
LIN {X 0,Y 425.359,Z 1204.891,A -85,B 0,C 180,E1 16451.837,E2 16451.837} C_VEL
LIN {X 0,Y 423.49,Z 1218.382,A -85,B 0,C 180,E1 16457.077,E2 16457.077} C_VEL
LIN {X 0,Y 422.686,Z 1227.659,A -85,B 0,C 180,E1 16462.792,E2 16462.792} C_VEL
LIN {X 0,Y 422.568,Z 1231.589,A -85,B 0,C 180,E1 16467.945,E2 16467.945} C_VEL
LIN {X 0,Y 422.54,Z 1231.589,A -85,B 0,C 180,E1 16472.055,E2 16472.055} C_VEL
LIN {X 0,Y 422.67,Z 1227.669,A -85,B 0,C 180,E1 16477.208,E2 16477.208} C_VEL
LIN {X 0,Y 423.502,Z 1218.398,A -85,B 0,C 180,E1 16482.922,E2 16482.922} C_VEL
LIN {X 0,Y 425.628,Z 1203.309,A -85,B 0,C 180,E1 16488.688,E2 16488.688} C_VEL
LIN {X 0,Y 429.685,Z 1183.727,A -85,B 0,C 180,E1 16494.015,E2 16494.015} C_VEL
LIN {X 0,Y 432.452,Z 1172.346,A -85,B 0,C 180,E1 16496.505,E2 16496.505} C_VEL
LIN {X 0,Y 431.04,Z 1163.37,A -85,B 0,C 180,E1 16498.493,E2 16498.493} C_VEL
LIN {X 0,Y 429.657,Z 1155.094,A -85,B 0,C 180,E1 16500.209,E2 16500.209} C_VEL
LIN {X 0,Y 429.949,Z 1153.772,A -85,B 0,C 180,E1 16500.44,E2 16500.44} C_VEL
LIN {X 0,Y 437.938,Z 1124.559,A -85,B 0,C 180,E1 16504.813,E2 16504.813} C_VEL
LIN {X 0,Y 447.231,Z 1089.311,A -85,B 0,C 180,E1 16508.82,E2 16508.82} C_VEL
LIN {X 0,Y 456.463,Z 1050.71,A -85,B 0,C 180,E1 16512.079,E2 16512.079} C_VEL
LIN {X 0,Y 465.01,Z 1007.136,A -85,B 0,C 180,E1 16514.722,E2 16514.722} C_VEL
LIN {X 0,Y 470.334,Z 968.519,A -85,B 0,C 180,E1 16516.383,E2 16516.383} C_VEL
LIN {X 0,Y 457.173,Z 934.775,A -85,B 0,C 180,E1 16519.432,E2 16519.432} C_VEL
LIN {X 0,Y 438.487,Z 900.379,A -85,B 0,C 180,E1 16523.098,E2 16523.098} C_VEL
LIN {X 0,Y 419.964,Z 871.697,A -85,B 0,C 180,E1 16527.079,E2 16527.079} C_VEL
LIN {X 0,Y 415.133,Z 864.887,A -85,B 0,C 180,E1 16528.224,E2 16528.224} C_VEL
LIN {X 0,Y 412.866,Z 860.37,A -85,B 0,C 180,E1 16528.823,E2 16528.823} C_VEL
LIN {X 0,Y 412.797,Z 859.31,A -85,B 0,C 180,E1 16529.081,E2 16529.081} C_VEL
LIN {X 0,Y 413.179,Z 859.31,A -85,B 0,C 180,E1 16536.469,E2 16536.469} C_VEL
LIN {X 0,Y 413.384,Z 859.31,A -85,B 0,C 180,E1 16542.949,E2 16542.949} C_VEL
LIN {X 0,Y 413.72,Z 859.31,A -85,B 0,C 180,E1 16549.448,E2 16549.448} C_VEL
LIN {X 0,Y 414.257,Z 859.31,A -85,B 0,C 180,E1 16555.803,E2 16555.803} C_VEL
LIN {X 0,Y 414.44,Z 859.31,A -85,B 0,C 180,E1 16562.092,E2 16562.092} C_VEL
LIN {X 0,Y 413.851,Z 859.31,A -85,B 0,C 180,E1 16568.665,E2 16568.665} C_VEL
LIN {X 0,Y 413.499,Z 859.31,A -85,B 0,C 180,E1 16574.857,E2 16574.857} C_VEL
LIN {X 0,Y 413.185,Z 859.31,A -85,B 0,C 180,E1 16581.505,E2 16581.505} C_VEL
LIN {X 0,Y 412.843,Z 859.31,A -85,B 0,C 180,E1 16588.488,E2 16588.488} C_VEL
LIN {X 0,Y 412.654,Z 859.31,A -85,B 0,C 180,E1 16593.409,E2 16593.409} C_VEL
LIN {X 0,Y 412.582,Z 859.872,A -85,B 0,C 180,E1 16597.196,E2 16597.196} C_VEL
LIN {X 0,Y 415.367,Z 865.327,A -85,B 0,C 180,E1 16597.913,E2 16597.913} C_VEL
LIN {X 0,Y 433.177,Z 891.26,A -85,B 0,C 180,E1 16601.804,E2 16601.804} C_VEL
LIN {X 0,Y 453.724,Z 925.758,A -85,B 0,C 180,E1 16605.668,E2 16605.668} C_VEL
LIN {X 0,Y 471.471,Z 962.269,A -85,B 0,C 180,E1 16608.839,E2 16608.839} C_VEL
LIN {X 0,Y 472.59,Z 968.11,A -85,B 0,C 180,E1 16609.163,E2 16609.163} C_VEL
LIN {X 0,Y 466.952,Z 1009.63,A -85,B 0,C 180,E1 16610.519,E2 16610.519} C_VEL
LIN {X 0,Y 459.602,Z 1047.755,A -85,B 0,C 180,E1 16612.522,E2 16612.522} C_VEL
LIN {X 0,Y 450.511,Z 1084.409,A -85,B 0,C 180,E1 16615.319,E2 16615.319} C_VEL
LIN {X 0,Y 441.26,Z 1116.249,A -85,B 0,C 180,E1 16618.709,E2 16618.709} C_VEL
LIN {X 0,Y 432.161,Z 1144.802,A -85,B 0,C 180,E1 16622.882,E2 16622.882} C_VEL
LIN {X 0,Y 425.09,Z 1167.243,A -85,B 0,C 180,E1 16627.368,E2 16627.368} C_VEL
LIN {X 0,Y 419.476,Z 1186.232,A -85,B 0,C 180,E1 16632.662,E2 16632.662} C_VEL
LIN {X 0,Y 416.206,Z 1200.059,A -85,B 0,C 180,E1 16638.449,E2 16638.449} C_VEL
LIN {X 0,Y 414.975,Z 1207.481,A -85,B 0,C 180,E1 16643.711,E2 16643.711} C_VEL
LIN {X 0,Y 414.664,Z 1210.226,A -85,B 0,C 180,E1 16647.906,E2 16647.906} C_VEL
LIN {X 0,Y 414.74,Z 1210.177,A -85,B 0,C 180,E1 16652.094,E2 16652.094} C_VEL
LIN {X 0,Y 415.164,Z 1206.226,A -85,B 0,C 180,E1 16657.34,E2 16657.34} C_VEL
LIN {X 0,Y 416.932,Z 1196.656,A -85,B 0,C 180,E1 16663.13,E2 16663.13} C_VEL
LIN {X 0,Y 420.936,Z 1180.952,A -85,B 0,C 180,E1 16668.904,E2 16668.904} C_VEL
LIN {X 0,Y 427.595,Z 1159.062,A -85,B 0,C 180,E1 16674.328,E2 16674.328} C_VEL
LIN {X 0,Y 435.797,Z 1133.417,A -85,B 0,C 180,E1 16678.845,E2 16678.845} C_VEL
LIN {X 0,Y 445.41,Z 1102.071,A -85,B 0,C 180,E1 16682.834,E2 16682.834} C_VEL
LIN {X 0,Y 454.712,Z 1067.851,A -85,B 0,C 180,E1 16685.969,E2 16685.969} C_VEL
LIN {X 0,Y 462.992,Z 1030.976,A -85,B 0,C 180,E1 16688.358,E2 16688.358} C_VEL
LIN {X 0,Y 469.579,Z 992.129,A -85,B 0,C 180,E1 16690.044,E2 16690.044} C_VEL
LIN {X 0,Y 472.363,Z 964.535,A -85,B 0,C 180,E1 16690.874,E2 16690.874} C_VEL
LIN {X 0,Y 454.785,Z 927.784,A -85,B 0,C 180,E1 16694.026,E2 16694.026} C_VEL
LIN {X 0,Y 434.686,Z 893.756,A -85,B 0,C 180,E1 16697.766,E2 16697.766} C_VEL
LIN {X 0,Y 415.542,Z 865.401,A -85,B 0,C 180,E1 16701.916,E2 16701.916} C_VEL
LIN {X 0,Y 412.679,Z 860.372,A -85,B 0,C 180,E1 16702.634,E2 16702.634} C_VEL
LIN {X 0,Y 412.573,Z 859.31,A -85,B 0,C 180,E1 16702.798,E2 16702.798} C_VEL
LIN {X 0,Y 412.715,Z 859.31,A -85,B 0,C 180,E1 16709.081,E2 16709.081} C_VEL
LIN {X 0,Y 413.028,Z 859.31,A -85,B 0,C 180,E1 16716.209,E2 16716.209} C_VEL
LIN {X 0,Y 413.22,Z 859.31,A -85,B 0,C 180,E1 16722.948,E2 16722.948} C_VEL
LIN {X 0,Y 413.775,Z 859.31,A -85,B 0,C 180,E1 16729.455,E2 16729.455} C_VEL
LIN {X 0,Y 414.264,Z 859.31,A -85,B 0,C 180,E1 16735.809,E2 16735.809} C_VEL
LIN {X 0,Y 414.445,Z 859.31,A -85,B 0,C 180,E1 16742.098,E2 16742.098} C_VEL
LIN {X 0,Y 413.841,Z 859.31,A -85,B 0,C 180,E1 16748.653,E2 16748.653} C_VEL
LIN {X 0,Y 413.508,Z 859.31,A -85,B 0,C 180,E1 16754.862,E2 16754.862} C_VEL
LIN {X 0,Y 413.216,Z 859.31,A -85,B 0,C 180,E1 16761.51,E2 16761.51} C_VEL
LIN {X 0,Y 412.867,Z 859.31,A -85,B 0,C 180,E1 16768.493,E2 16768.493} C_VEL
LIN {X 0,Y 412.764,Z 859.734,A -85,B 0,C 180,E1 16771.182,E2 16771.182} C_VEL
LIN {X 0,Y 415.225,Z 865.068,A -85,B 0,C 180,E1 16771.844,E2 16771.844} C_VEL
LIN {X 0,Y 425.513,Z 879.842,A -85,B 0,C 180,E1 16774.211,E2 16774.211} C_VEL
LIN {X 0,Y 447.304,Z 915.618,A -85,B 0,C 180,E1 16778.647,E2 16778.647} C_VEL
LIN {X 0,Y 464.278,Z 951.615,A -85,B 0,C 180,E1 16782.143,E2 16782.143} C_VEL
LIN {X 0,Y 470.499,Z 969.982,A -85,B 0,C 180,E1 16783.727,E2 16783.727} C_VEL
LIN {X 0,Y 464.175,Z 1011.277,A -85,B 0,C 180,E1 16785.506,E2 16785.506} C_VEL
LIN {X 0,Y 456.103,Z 1052.12,A -85,B 0,C 180,E1 16788.04,E2 16788.04} C_VEL
LIN {X 0,Y 446.722,Z 1091.239,A -85,B 0,C 180,E1 16791.377,E2 16791.377} C_VEL
LIN {X 0,Y 437.404,Z 1126.44,A -85,B 0,C 180,E1 16795.439,E2 16795.439} C_VEL
LIN {X 0,Y 428.694,Z 1158.24,A -85,B 0,C 180,E1 16800.34,E2 16800.34} C_VEL
LIN {X 0,Y 422.151,Z 1183.785,A -85,B 0,C 180,E1 16805.62,E2 16805.62} C_VEL
LIN {X 0,Y 417.934,Z 1203.04,A -85,B 0,C 180,E1 16810.955,E2 16810.955} C_VEL
LIN {X 0,Y 415.653,Z 1218.161,A -85,B 0,C 180,E1 16816.829,E2 16816.829} C_VEL
LIN {X 0,Y 414.791,Z 1227.449,A -85,B 0,C 180,E1 16822.654,E2 16822.654} C_VEL
LIN {X 0,Y 414.661,Z 1231.386,A -85,B 0,C 180,E1 16827.906,E2 16827.906} C_VEL
LIN {X 0,Y 414.635,Z 1231.387,A -85,B 0,C 180,E1 16832.094,E2 16832.094} C_VEL
LIN {X 0,Y 414.773,Z 1227.46,A -85,B 0,C 180,E1 16837.346,E2 16837.346} C_VEL
LIN {X 0,Y 415.667,Z 1218.179,A -85,B 0,C 180,E1 16843.17,E2 16843.17} C_VEL
LIN {X 0,Y 417.916,Z 1203.069,A -85,B 0,C 180,E1 16849.046,E2 16849.046} C_VEL
LIN {X 0,Y 422.119,Z 1183.824,A -85,B 0,C 180,E1 16854.382,E2 16854.382} C_VEL
LIN {X 0,Y 428.62,Z 1158.306,A -85,B 0,C 180,E1 16859.665,E2 16859.665} C_VEL
LIN {X 0,Y 429.949,Z 1153.772,A -85,B 0,C 180,E1 16860.44,E2 16860.44} C_VEL
LIN {X 0,Y 429.14,Z 1143.722,A -85,B 0,C 180,E1 16862.355,E2 16862.355} C_VEL
LIN {X 0,Y 428.358,Z 1134.543,A -85,B 0,C 180,E1 16863.995,E2 16863.995} C_VEL
LIN {X 0,Y 428.744,Z 1133.07,A -85,B 0,C 180,E1 16864.208,E2 16864.208} C_VEL
LIN {X 0,Y 437.955,Z 1099.849,A -85,B 0,C 180,E1 16868.346,E2 16868.346} C_VEL
LIN {X 0,Y 447.362,Z 1063.132,A -85,B 0,C 180,E1 16871.78,E2 16871.78} C_VEL
LIN {X 0,Y 456.633,Z 1020.682,A -85,B 0,C 180,E1 16874.658,E2 16874.658} C_VEL
LIN {X 0,Y 464.208,Z 975.89,A -85,B 0,C 180,E1 16876.736,E2 16876.736} C_VEL
LIN {X 0,Y 464.028,Z 970.383,A -85,B 0,C 180,E1 16877.036,E2 16877.036} C_VEL
LIN {X 0,Y 451.164,Z 937.28,A -85,B 0,C 180,E1 16880.151,E2 16880.151} C_VEL
LIN {X 0,Y 433.401,Z 904.381,A -85,B 0,C 180,E1 16883.8,E2 16883.8} C_VEL
LIN {X 0,Y 415.534,Z 876.766,A -85,B 0,C 180,E1 16887.774,E2 16887.774} C_VEL
LIN {X 0,Y 407.737,Z 865.418,A -85,B 0,C 180,E1 16889.729,E2 16889.729} C_VEL
LIN {X 0,Y 405.026,Z 860.923,A -85,B 0,C 180,E1 16890.469,E2 16890.469} C_VEL
LIN {X 0,Y 404.883,Z 859.31,A -85,B 0,C 180,E1 16890.718,E2 16890.718} C_VEL
LIN {X 0,Y 405.138,Z 859.31,A -85,B 0,C 180,E1 16895.71,E2 16895.71} C_VEL
LIN {X 0,Y 405.45,Z 859.31,A -85,B 0,C 180,E1 16902.605,E2 16902.605} C_VEL
LIN {X 0,Y 405.779,Z 859.31,A -85,B 0,C 180,E1 16909.239,E2 16909.239} C_VEL
LIN {X 0,Y 406.337,Z 859.31,A -85,B 0,C 180,E1 16915.721,E2 16915.721} C_VEL
LIN {X 0,Y 406.531,Z 859.31,A -85,B 0,C 180,E1 16922.133,E2 16922.133} C_VEL
LIN {X 0,Y 405.98,Z 859.31,A -85,B 0,C 180,E1 16928.581,E2 16928.581} C_VEL
LIN {X 0,Y 405.557,Z 859.31,A -85,B 0,C 180,E1 16935.154,E2 16935.154} C_VEL
LIN {X 0,Y 405.224,Z 859.31,A -85,B 0,C 180,E1 16941.949,E2 16941.949} C_VEL
LIN {X 0,Y 404.838,Z 859.31,A -85,B 0,C 180,E1 16949.105,E2 16949.105} C_VEL
LIN {X 0,Y 404.602,Z 859.31,A -85,B 0,C 180,E1 16955.465,E2 16955.465} C_VEL
LIN {X 0,Y 406.606,Z 864.53,A -85,B 0,C 180,E1 16956.071,E2 16956.071} C_VEL
LIN {X 0,Y 409.714,Z 868.238,A -85,B 0,C 180,E1 16956.843,E2 16956.843} C_VEL
LIN {X 0,Y 429.51,Z 897.377,A -85,B 0,C 180,E1 16961.342,E2 16961.342} C_VEL
LIN {X 0,Y 449.563,Z 931.39,A -85,B 0,C 180,E1 16965.21,E2 16965.21} C_VEL
LIN {X 0,Y 466.229,Z 966.683,A -85,B 0,C 180,E1 16968.355,E2 16968.355} C_VEL
LIN {X 0,Y 466.003,Z 976.351,A -85,B 0,C 180,E1 16968.713,E2 16968.713} C_VEL
LIN {X 0,Y 459.934,Z 1016.609,A -85,B 0,C 180,E1 16970.18,E2 16970.18} C_VEL
LIN {X 0,Y 452.269,Z 1053.093,A -85,B 0,C 180,E1 16972.234,E2 16972.234} C_VEL
LIN {X 0,Y 443.453,Z 1086.853,A -85,B 0,C 180,E1 16974.928,E2 16974.928} C_VEL
LIN {X 0,Y 434.474,Z 1116.588,A -85,B 0,C 180,E1 16978.163,E2 16978.163} C_VEL
LIN {X 0,Y 425.063,Z 1145.082,A -85,B 0,C 180,E1 16982.391,E2 16982.391} C_VEL
LIN {X 0,Y 417.393,Z 1168.471,A -85,B 0,C 180,E1 16987.192,E2 16987.192} C_VEL
LIN {X 0,Y 411.868,Z 1186.454,A -85,B 0,C 180,E1 16992.331,E2 16992.331} C_VEL
LIN {X 0,Y 408.394,Z 1200.269,A -85,B 0,C 180,E1 16998.225,E2 16998.225} C_VEL
LIN {X 0,Y 407.097,Z 1207.686,A -85,B 0,C 180,E1 17003.589,E2 17003.589} C_VEL
LIN {X 0,Y 406.778,Z 1210.428,A -85,B 0,C 180,E1 17007.865,E2 17007.865} C_VEL
LIN {X 0,Y 406.845,Z 1210.379,A -85,B 0,C 180,E1 17012.135,E2 17012.135} C_VEL
LIN {X 0,Y 407.289,Z 1206.432,A -85,B 0,C 180,E1 17017.482,E2 17017.482} C_VEL
LIN {X 0,Y 409.161,Z 1196.872,A -85,B 0,C 180,E1 17023.384,E2 17023.384} C_VEL
LIN {X 0,Y 412.844,Z 1182.848,A -85,B 0,C 180,E1 17028.733,E2 17028.733} C_VEL
LIN {X 0,Y 419.135,Z 1162.863,A -85,B 0,C 180,E1 17033.999,E2 17033.999} C_VEL
LIN {X 0,Y 427.263,Z 1138.456,A -85,B 0,C 180,E1 17038.606,E2 17038.606} C_VEL
LIN {X 0,Y 436.533,Z 1109.835,A -85,B 0,C 180,E1 17042.55,E2 17042.55} C_VEL
LIN {X 0,Y 445.773,Z 1078.182,A -85,B 0,C 180,E1 17045.75,E2 17045.75} C_VEL
LIN {X 0,Y 454.561,Z 1042.729,A -85,B 0,C 180,E1 17048.331,E2 17048.331} C_VEL
LIN {X 0,Y 461.893,Z 1004.778,A -85,B 0,C 180,E1 17050.231,E2 17050.231} C_VEL
LIN {X 0,Y 466.377,Z 967.287,A -85,B 0,C 180,E1 17051.49,E2 17051.49} C_VEL
LIN {X 0,Y 449.725,Z 931.815,A -85,B 0,C 180,E1 17054.639,E2 17054.639} C_VEL
LIN {X 0,Y 429.864,Z 897.904,A -85,B 0,C 180,E1 17058.464,E2 17058.464} C_VEL
LIN {X 0,Y 411.654,Z 871.234,A -85,B 0,C 180,E1 17062.533,E2 17062.533} C_VEL
LIN {X 0,Y 407.464,Z 865.363,A -85,B 0,C 180,E1 17063.575,E2 17063.575} C_VEL
LIN {X 0,Y 404.714,Z 860.425,A -85,B 0,C 180,E1 17064.324,E2 17064.324} C_VEL
LIN {X 0,Y 404.635,Z 859.31,A -85,B 0,C 180,E1 17064.389,E2 17064.389} C_VEL
LIN {X 0,Y 404.843,Z 859.31,A -85,B 0,C 180,E1 17070.896,E2 17070.896} C_VEL
LIN {X 0,Y 405.044,Z 859.31,A -85,B 0,C 180,E1 17075.71,E2 17075.71} C_VEL
LIN {X 0,Y 405.307,Z 859.31,A -85,B 0,C 180,E1 17082.605,E2 17082.605} C_VEL
LIN {X 0,Y 405.823,Z 859.31,A -85,B 0,C 180,E1 17089.246,E2 17089.246} C_VEL
LIN {X 0,Y 406.345,Z 859.31,A -85,B 0,C 180,E1 17095.727,E2 17095.727} C_VEL
LIN {X 0,Y 406.536,Z 859.31,A -85,B 0,C 180,E1 17102.138,E2 17102.138} C_VEL
LIN {X 0,Y 405.969,Z 859.31,A -85,B 0,C 180,E1 17108.587,E2 17108.587} C_VEL
LIN {X 0,Y 405.566,Z 859.31,A -85,B 0,C 180,E1 17115.16,E2 17115.16} C_VEL
LIN {X 0,Y 405.275,Z 859.31,A -85,B 0,C 180,E1 17121.953,E2 17121.953} C_VEL
LIN {X 0,Y 404.868,Z 859.31,A -85,B 0,C 180,E1 17129.109,E2 17129.109} C_VEL
LIN {X 0,Y 404.856,Z 859.685,A -85,B 0,C 180,E1 17129.498,E2 17129.498} C_VEL
LIN {X 0,Y 407.026,Z 864.794,A -85,B 0,C 180,E1 17130.144,E2 17130.144} C_VEL
LIN {X 0,Y 409.758,Z 868.191,A -85,B 0,C 180,E1 17130.835,E2 17130.835} C_VEL
LIN {X 0,Y 426.613,Z 893.453,A -85,B 0,C 180,E1 17134.796,E2 17134.796} C_VEL
LIN {X 0,Y 445.94,Z 927.014,A -85,B 0,C 180,E1 17138.788,E2 17138.788} C_VEL
LIN {X 0,Y 461.094,Z 961.679,A -85,B 0,C 180,E1 17142.183,E2 17142.183} C_VEL
LIN {X 0,Y 464.264,Z 973.807,A -85,B 0,C 180,E1 17143.186,E2 17143.186} C_VEL
LIN {X 0,Y 457.408,Z 1015.849,A -85,B 0,C 180,E1 17145.086,E2 17145.086} C_VEL
LIN {X 0,Y 449.057,Z 1055.827,A -85,B 0,C 180,E1 17147.675,E2 17147.675} C_VEL
LIN {X 0,Y 439.839,Z 1092.711,A -85,B 0,C 180,E1 17150.913,E2 17150.913} C_VEL
LIN {X 0,Y 430.144,Z 1128.008,A -85,B 0,C 180,E1 17155.079,E2 17155.079} C_VEL
LIN {X 0,Y 421.201,Z 1159.433,A -85,B 0,C 180,E1 17160.055,E2 17160.055} C_VEL
LIN {X 0,Y 414.204,Z 1185.776,A -85,B 0,C 180,E1 17165.697,E2 17165.697} C_VEL
LIN {X 0,Y 409.665,Z 1206.013,A -85,B 0,C 180,E1 17171.675,E2 17171.675} C_VEL
LIN {X 0,Y 407.578,Z 1219.975,A -85,B 0,C 180,E1 17177.656,E2 17177.656} C_VEL
LIN {X 0,Y 406.85,Z 1228.392,A -85,B 0,C 180,E1 17183.584,E2 17183.584} C_VEL
LIN {X 0,Y 406.773,Z 1231.185,A -85,B 0,C 180,E1 17187.865,E2 17187.865} C_VEL
LIN {X 0,Y 406.751,Z 1231.186,A -85,B 0,C 180,E1 17192.135,E2 17192.135} C_VEL
LIN {X 0,Y 406.897,Z 1227.252,A -85,B 0,C 180,E1 17197.489,E2 17197.489} C_VEL
LIN {X 0,Y 407.815,Z 1217.96,A -85,B 0,C 180,E1 17203.428,E2 17203.428} C_VEL
LIN {X 0,Y 410.251,Z 1202.83,A -85,B 0,C 180,E1 17209.416,E2 17209.416} C_VEL
LIN {X 0,Y 414.635,Z 1183.554,A -85,B 0,C 180,E1 17214.851,E2 17214.851} C_VEL
LIN {X 0,Y 421.522,Z 1157.995,A -85,B 0,C 180,E1 17220.217,E2 17220.217} C_VEL
LIN {X 0,Y 428.744,Z 1133.07,A -85,B 0,C 180,E1 17224.208,E2 17224.208} C_VEL
LIN {X 0,Y 428.998,Z 1124.698,A -85,B 0,C 180,E1 17225.559,E2 17225.559} C_VEL
LIN {X 0,Y 427.987,Z 1111.957,A -85,B 0,C 180,E1 17227.587,E2 17227.587} C_VEL
LIN {X 0,Y 428.419,Z 1110.347,A -85,B 0,C 180,E1 17227.78,E2 17227.78} C_VEL
LIN {X 0,Y 438.336,Z 1074.505,A -85,B 0,C 180,E1 17231.466,E2 17231.466} C_VEL
LIN {X 0,Y 447.821,Z 1035.029,A -85,B 0,C 180,E1 17234.461,E2 17234.461} C_VEL
LIN {X 0,Y 455.908,Z 993.029,A -85,B 0,C 180,E1 17236.727,E2 17236.727} C_VEL
LIN {X 0,Y 458.228,Z 973.789,A -85,B 0,C 180,E1 17237.571,E2 17237.571} C_VEL
LIN {X 0,Y 445.643,Z 940.703,A -85,B 0,C 180,E1 17240.794,E2 17240.794} C_VEL
LIN {X 0,Y 428.031,Z 907.68,A -85,B 0,C 180,E1 17244.597,E2 17244.597} C_VEL
LIN {X 0,Y 409.038,Z 878.264,A -85,B 0,C 180,E1 17249.034,E2 17249.034} C_VEL
LIN {X 0,Y 399.876,Z 865.444,A -85,B 0,C 180,E1 17251.485,E2 17251.485} C_VEL
LIN {X 0,Y 397.171,Z 860.994,A -85,B 0,C 180,E1 17252.289,E2 17252.289} C_VEL
LIN {X 0,Y 396.999,Z 859.31,A -85,B 0,C 180,E1 17252.432,E2 17252.432} C_VEL
LIN {X 0,Y 397.299,Z 859.31,A -85,B 0,C 180,E1 17257.583,E2 17257.583} C_VEL
LIN {X 0,Y 397.59,Z 859.31,A -85,B 0,C 180,E1 17264.528,E2 17264.528} C_VEL
LIN {X 0,Y 398.071,Z 859.31,A -85,B 0,C 180,E1 17271.773,E2 17271.773} C_VEL
LIN {X 0,Y 398.561,Z 859.31,A -85,B 0,C 180,E1 17277.819,E2 17277.819} C_VEL
LIN {X 0,Y 398.619,Z 859.31,A -85,B 0,C 180,E1 17282.175,E2 17282.175} C_VEL
LIN {X 0,Y 398.046,Z 859.31,A -85,B 0,C 180,E1 17288.753,E2 17288.753} C_VEL
LIN {X 0,Y 397.608,Z 859.31,A -85,B 0,C 180,E1 17295.465,E2 17295.465} C_VEL
LIN {X 0,Y 397.239,Z 859.31,A -85,B 0,C 180,E1 17302.414,E2 17302.414} C_VEL
LIN {X 0,Y 396.913,Z 859.31,A -85,B 0,C 180,E1 17309.743,E2 17309.743} C_VEL
LIN {X 0,Y 396.716,Z 859.438,A -85,B 0,C 180,E1 17313.631,E2 17313.631} C_VEL
LIN {X 0,Y 398.841,Z 864.69,A -85,B 0,C 180,E1 17314.315,E2 17314.315} C_VEL
LIN {X 0,Y 401.763,Z 868.022,A -85,B 0,C 180,E1 17315.101,E2 17315.101} C_VEL
LIN {X 0,Y 418.725,Z 892.454,A -85,B 0,C 180,E1 17319.297,E2 17319.297} C_VEL
LIN {X 0,Y 438.378,Z 924.309,A -85,B 0,C 180,E1 17323.409,E2 17323.409} C_VEL
LIN {X 0,Y 455.888,Z 958.774,A -85,B 0,C 180,E1 17326.796,E2 17326.796} C_VEL
LIN {X 0,Y 460.803,Z 972.356,A -85,B 0,C 180,E1 17327.921,E2 17327.921} C_VEL
LIN {X 0,Y 454.962,Z 1011.456,A -85,B 0,C 180,E1 17329.263,E2 17329.263} C_VEL
LIN {X 0,Y 447.087,Z 1049.453,A -85,B 0,C 180,E1 17331.328,E2 17331.328} C_VEL
LIN {X 0,Y 438.084,Z 1083.63,A -85,B 0,C 180,E1 17333.984,E2 17333.984} C_VEL
LIN {X 0,Y 428.367,Z 1115.048,A -85,B 0,C 180,E1 17337.354,E2 17337.354} C_VEL
LIN {X 0,Y 418.563,Z 1143.944,A -85,B 0,C 180,E1 17341.631,E2 17341.631} C_VEL
LIN {X 0,Y 410.239,Z 1168.114,A -85,B 0,C 180,E1 17346.606,E2 17346.606} C_VEL
LIN {X 0,Y 404.243,Z 1186.676,A -85,B 0,C 180,E1 17351.986,E2 17351.986} C_VEL
LIN {X 0,Y 400.606,Z 1200.478,A -85,B 0,C 180,E1 17357.993,E2 17357.993} C_VEL
LIN {X 0,Y 399.214,Z 1207.891,A -85,B 0,C 180,E1 17363.462,E2 17363.462} C_VEL
LIN {X 0,Y 398.879,Z 1210.63,A -85,B 0,C 180,E1 17367.823,E2 17367.823} C_VEL
LIN {X 0,Y 398.945,Z 1210.582,A -85,B 0,C 180,E1 17372.177,E2 17372.177} C_VEL
LIN {X 0,Y 399.425,Z 1206.638,A -85,B 0,C 180,E1 17377.63,E2 17377.63} C_VEL
LIN {X 0,Y 401.398,Z 1197.087,A -85,B 0,C 180,E1 17383.647,E2 17383.647} C_VEL
LIN {X 0,Y 405.831,Z 1181.414,A -85,B 0,C 180,E1 17389.636,E2 17389.636} C_VEL
LIN {X 0,Y 413.104,Z 1159.608,A -85,B 0,C 180,E1 17395.24,E2 17395.24} C_VEL
LIN {X 0,Y 421.891,Z 1134.065,A -85,B 0,C 180,E1 17399.891,E2 17399.891} C_VEL
LIN {X 0,Y 432.157,Z 1102.884,A -85,B 0,C 180,E1 17403.975,E2 17403.975} C_VEL
LIN {X 0,Y 442.036,Z 1068.943,A -85,B 0,C 180,E1 17407.17,E2 17407.17} C_VEL
LIN {X 0,Y 451.042,Z 1031.257,A -85,B 0,C 180,E1 17409.666,E2 17409.666} C_VEL
LIN {X 0,Y 458.187,Z 991.486,A -85,B 0,C 180,E1 17411.409,E2 17411.409} C_VEL
LIN {X 0,Y 460.467,Z 969.977,A -85,B 0,C 180,E1 17412.103,E2 17412.103} C_VEL
LIN {X 0,Y 444.098,Z 934.702,A -85,B 0,C 180,E1 17415.38,E2 17415.38} C_VEL
LIN {X 0,Y 424.775,Z 901.753,A -85,B 0,C 180,E1 17419.238,E2 17419.238} C_VEL
LIN {X 0,Y 405.2,Z 872.658,A -85,B 0,C 180,E1 17423.847,E2 17423.847} C_VEL
LIN {X 0,Y 399.572,Z 865.382,A -85,B 0,C 180,E1 17425.345,E2 17425.345} C_VEL
LIN {X 0,Y 396.796,Z 860.378,A -85,B 0,C 180,E1 17426.17,E2 17426.17} C_VEL
LIN {X 0,Y 396.71,Z 859.31,A -85,B 0,C 180,E1 17426.435,E2 17426.435} C_VEL
LIN {X 0,Y 396.954,Z 859.31,A -85,B 0,C 180,E1 17432.748,E2 17432.748} C_VEL
LIN {X 0,Y 397.289,Z 859.31,A -85,B 0,C 180,E1 17439.933,E2 17439.933} C_VEL
LIN {X 0,Y 397.673,Z 859.31,A -85,B 0,C 180,E1 17446.791,E2 17446.791} C_VEL
LIN {X 0,Y 398.257,Z 859.31,A -85,B 0,C 180,E1 17453.45,E2 17453.45} C_VEL
LIN {X 0,Y 398.746,Z 859.31,A -85,B 0,C 180,E1 17460.003,E2 17460.003} C_VEL
LIN {X 0,Y 398.236,Z 859.31,A -85,B 0,C 180,E1 17466.556,E2 17466.556} C_VEL
LIN {X 0,Y 397.77,Z 859.31,A -85,B 0,C 180,E1 17473.212,E2 17473.212} C_VEL
LIN {X 0,Y 397.428,Z 859.31,A -85,B 0,C 180,E1 17480.066,E2 17480.066} C_VEL
LIN {X 0,Y 396.983,Z 859.31,A -85,B 0,C 180,E1 17487.256,E2 17487.256} C_VEL
LIN {X 0,Y 396.976,Z 859.31,A -85,B 0,C 180,E1 17487.645,E2 17487.645} C_VEL
LIN {X 0,Y 399.021,Z 864.652,A -85,B 0,C 180,E1 17488.344,E2 17488.344} C_VEL
LIN {X 0,Y 401.879,Z 867.968,A -85,B 0,C 180,E1 17489.116,E2 17489.116} C_VEL
LIN {X 0,Y 419.262,Z 893.704,A -85,B 0,C 180,E1 17493.489,E2 17493.489} C_VEL
LIN {X 0,Y 438.816,Z 927.035,A -85,B 0,C 180,E1 17497.737,E2 17497.737} C_VEL
LIN {X 0,Y 453.899,Z 961.048,A -85,B 0,C 180,E1 17501.239,E2 17501.239} C_VEL
LIN {X 0,Y 458.319,Z 976.077,A -85,B 0,C 180,E1 17502.58,E2 17502.58} C_VEL
LIN {X 0,Y 450.669,Z 1020.447,A -85,B 0,C 180,E1 17504.655,E2 17504.655} C_VEL
LIN {X 0,Y 441.451,Z 1062.047,A -85,B 0,C 180,E1 17507.497,E2 17507.497} C_VEL
LIN {X 0,Y 431.971,Z 1097.976,A -85,B 0,C 180,E1 17510.845,E2 17510.845} C_VEL
LIN {X 0,Y 422.861,Z 1129.605,A -85,B 0,C 180,E1 17514.726,E2 17514.726} C_VEL
LIN {X 0,Y 413.682,Z 1160.532,A -85,B 0,C 180,E1 17519.758,E2 17519.758} C_VEL
LIN {X 0,Y 406.493,Z 1186.587,A -85,B 0,C 180,E1 17525.499,E2 17525.499} C_VEL
LIN {X 0,Y 401.706,Z 1207.341,A -85,B 0,C 180,E1 17531.868,E2 17531.868} C_VEL
LIN {X 0,Y 399.624,Z 1220.772,A -85,B 0,C 180,E1 17537.962,E2 17537.962} C_VEL
LIN {X 0,Y 398.952,Z 1228.186,A -85,B 0,C 180,E1 17543.457,E2 17543.457} C_VEL
LIN {X 0,Y 398.865,Z 1230.982,A -85,B 0,C 180,E1 17547.823,E2 17547.823} C_VEL
LIN {X 0,Y 398.845,Z 1230.984,A -85,B 0,C 180,E1 17552.177,E2 17552.177} C_VEL
LIN {X 0,Y 399.02,Z 1227.044,A -85,B 0,C 180,E1 17557.638,E2 17557.638} C_VEL
LIN {X 0,Y 399.984,Z 1217.743,A -85,B 0,C 180,E1 17563.696,E2 17563.696} C_VEL
LIN {X 0,Y 402.605,Z 1202.52,A -85,B 0,C 180,E1 17569.826,E2 17569.826} C_VEL
LIN {X 0,Y 407.22,Z 1183.287,A -85,B 0,C 180,E1 17575.336,E2 17575.336} C_VEL
LIN {X 0,Y 414.504,Z 1157.688,A -85,B 0,C 180,E1 17580.783,E2 17580.783} C_VEL
LIN {X 0,Y 423.911,Z 1126.184,A -85,B 0,C 180,E1 17585.764,E2 17585.764} C_VEL
LIN {X 0,Y 428.419,Z 1110.347,A -85,B 0,C 180,E1 17587.78,E2 17587.78} C_VEL
LIN {X 0,Y 428.875,Z 1098.186,A -85,B 0,C 180,E1 17589.462,E2 17589.462} C_VEL
LIN {X 0,Y 429.091,Z 1085.587,A -85,B 0,C 180,E1 17591.097,E2 17591.097} C_VEL
LIN {X 0,Y 438.84,Z 1048.314,A -85,B 0,C 180,E1 17594.242,E2 17594.242} C_VEL
LIN {X 0,Y 447.659,Z 1006.814,A -85,B 0,C 180,E1 17596.787,E2 17596.787} C_VEL
LIN {X 0,Y 452.333,Z 976.719,A -85,B 0,C 180,E1 17598.164,E2 17598.164} C_VEL
LIN {X 0,Y 440.327,Z 944.446,A -85,B 0,C 180,E1 17601.419,E2 17601.419} C_VEL
LIN {X 0,Y 423.757,Z 912.862,A -85,B 0,C 180,E1 17605.182,E2 17605.182} C_VEL
LIN {X 0,Y 405.606,Z 884.431,A -85,B 0,C 180,E1 17609.553,E2 17609.553} C_VEL
LIN {X 0,Y 396.228,Z 871.408,A -85,B 0,C 180,E1 17612.138,E2 17612.138} C_VEL
LIN {X 0,Y 392.5,Z 865.806,A -85,B 0,C 180,E1 17613.27,E2 17613.27} C_VEL
LIN {X 0,Y 389.304,Z 860.773,A -85,B 0,C 180,E1 17614.299,E2 17614.299} C_VEL
LIN {X 0,Y 389.151,Z 859.31,A -85,B 0,C 180,E1 17614.407,E2 17614.407} C_VEL
LIN {X 0,Y 389.452,Z 859.31,A -85,B 0,C 180,E1 17619.504,E2 17619.504} C_VEL
LIN {X 0,Y 389.806,Z 859.31,A -85,B 0,C 180,E1 17626.513,E2 17626.513} C_VEL
LIN {X 0,Y 390.322,Z 859.31,A -85,B 0,C 180,E1 17633.311,E2 17633.311} C_VEL
LIN {X 0,Y 390.863,Z 859.31,A -85,B 0,C 180,E1 17639.997,E2 17639.997} C_VEL
LIN {X 0,Y 390.326,Z 859.31,A -85,B 0,C 180,E1 17646.683,E2 17646.683} C_VEL
LIN {X 0,Y 389.81,Z 859.31,A -85,B 0,C 180,E1 17653.637,E2 17653.637} C_VEL
LIN {X 0,Y 389.38,Z 859.31,A -85,B 0,C 180,E1 17660.938,E2 17660.938} C_VEL
LIN {X 0,Y 389.01,Z 859.31,A -85,B 0,C 180,E1 17667.856,E2 17667.856} C_VEL
LIN {X 0,Y 388.867,Z 859.979,A -85,B 0,C 180,E1 17671.63,E2 17671.63} C_VEL
LIN {X 0,Y 391.367,Z 865.088,A -85,B 0,C 180,E1 17672.473,E2 17672.473} C_VEL
LIN {X 0,Y 394.103,Z 868.234,A -85,B 0,C 180,E1 17673.278,E2 17673.278} C_VEL
LIN {X 0,Y 411.381,Z 892.704,A -85,B 0,C 180,E1 17677.887,E2 17677.887} C_VEL
LIN {X 0,Y 431.381,Z 924.615,A -85,B 0,C 180,E1 17682.31,E2 17682.31} C_VEL
LIN {X 0,Y 449.251,Z 959.668,A -85,B 0,C 180,E1 17685.94,E2 17685.94} C_VEL
LIN {X 0,Y 454.94,Z 974.98,A -85,B 0,C 180,E1 17687.291,E2 17687.291} C_VEL
LIN {X 0,Y 448.634,Z 1014.784,A -85,B 0,C 180,E1 17688.725,E2 17688.725} C_VEL
LIN {X 0,Y 440.45,Z 1052.133,A -85,B 0,C 180,E1 17690.831,E2 17690.831} C_VEL
LIN {X 0,Y 431.17,Z 1085.77,A -85,B 0,C 180,E1 17693.529,E2 17693.529} C_VEL
LIN {X 0,Y 421.046,Z 1117.258,A -85,B 0,C 180,E1 17697.021,E2 17697.021} C_VEL
LIN {X 0,Y 410.995,Z 1145.637,A -85,B 0,C 180,E1 17701.361,E2 17701.361} C_VEL
LIN {X 0,Y 402.506,Z 1169.401,A -85,B 0,C 180,E1 17706.423,E2 17706.423} C_VEL
LIN {X 0,Y 396.656,Z 1186.896,A -85,B 0,C 180,E1 17711.63,E2 17711.63} C_VEL
LIN {X 0,Y 392.818,Z 1200.687,A -85,B 0,C 180,E1 17717.751,E2 17717.751} C_VEL
LIN {X 0,Y 391.344,Z 1208.096,A -85,B 0,C 180,E1 17723.33,E2 17723.33} C_VEL
LIN {X 0,Y 391.002,Z 1210.832,A -85,B 0,C 180,E1 17727.779,E2 17727.779} C_VEL
LIN {X 0,Y 391.062,Z 1210.785,A -85,B 0,C 180,E1 17732.221,E2 17732.221} C_VEL
LIN {X 0,Y 391.569,Z 1206.843,A -85,B 0,C 180,E1 17737.785,E2 17737.785} C_VEL
LIN {X 0,Y 393.664,Z 1197.301,A -85,B 0,C 180,E1 17743.921,E2 17743.921} C_VEL
LIN {X 0,Y 398.281,Z 1181.645,A -85,B 0,C 180,E1 17750.024,E2 17750.024} C_VEL
LIN {X 0,Y 405.878,Z 1159.876,A -85,B 0,C 180,E1 17755.722,E2 17755.722} C_VEL
LIN {X 0,Y 415.579,Z 1132.68,A -85,B 0,C 180,E1 17760.696,E2 17760.696} C_VEL
LIN {X 0,Y 425.944,Z 1102.159,A -85,B 0,C 180,E1 17764.695,E2 17764.695} C_VEL
LIN {X 0,Y 436.174,Z 1067.965,A -85,B 0,C 180,E1 17767.914,E2 17767.914} C_VEL
LIN {X 0,Y 445.258,Z 1030.98,A -85,B 0,C 180,E1 17770.366,E2 17770.366} C_VEL
LIN {X 0,Y 452.602,Z 991.101,A -85,B 0,C 180,E1 17772.119,E2 17772.119} C_VEL
LIN {X 0,Y 454.491,Z 972.543,A -85,B 0,C 180,E1 17772.753,E2 17772.753} C_VEL
LIN {X 0,Y 438.545,Z 937.739,A -85,B 0,C 180,E1 17776.133,E2 17776.133} C_VEL
LIN {X 0,Y 420.478,Z 906.837,A -85,B 0,C 180,E1 17779.87,E2 17779.87} C_VEL
LIN {X 0,Y 402.028,Z 879.174,A -85,B 0,C 180,E1 17784.35,E2 17784.35} C_VEL
LIN {X 0,Y 392.186,Z 865.756,A -85,B 0,C 180,E1 17787.134,E2 17787.134} C_VEL
LIN {X 0,Y 389.056,Z 861.109,A -85,B 0,C 180,E1 17788.118,E2 17788.118} C_VEL
LIN {X 0,Y 388.853,Z 859.31,A -85,B 0,C 180,E1 17788.301,E2 17788.301} C_VEL
LIN {X 0,Y 389.105,Z 859.31,A -85,B 0,C 180,E1 17794.646,E2 17794.646} C_VEL
LIN {X 0,Y 389.412,Z 859.31,A -85,B 0,C 180,E1 17801.871,E2 17801.871} C_VEL
LIN {X 0,Y 389.933,Z 859.31,A -85,B 0,C 180,E1 17808.802,E2 17808.802} C_VEL
LIN {X 0,Y 390.528,Z 859.31,A -85,B 0,C 180,E1 17815.553,E2 17815.553} C_VEL
LIN {X 0,Y 390.867,Z 859.31,A -85,B 0,C 180,E1 17820.003,E2 17820.003} C_VEL
LIN {X 0,Y 390.322,Z 859.31,A -85,B 0,C 180,E1 17826.689,E2 17826.689} C_VEL
LIN {X 0,Y 389.801,Z 859.31,A -85,B 0,C 180,E1 17833.629,E2 17833.629} C_VEL
LIN {X 0,Y 389.416,Z 859.31,A -85,B 0,C 180,E1 17840.95,E2 17840.95} C_VEL
LIN {X 0,Y 389.111,Z 859.31,A -85,B 0,C 180,E1 17845.651,E2 17845.651} C_VEL
LIN {X 0,Y 390.994,Z 864.486,A -85,B 0,C 180,E1 17846.35,E2 17846.35} C_VEL
LIN {X 0,Y 394.242,Z 868.182,A -85,B 0,C 180,E1 17847.317,E2 17847.317} C_VEL
LIN {X 0,Y 411.239,Z 892.813,A -85,B 0,C 180,E1 17851.925,E2 17851.925} C_VEL
LIN {X 0,Y 429.779,Z 923.608,A -85,B 0,C 180,E1 17856.206,E2 17856.206} C_VEL
LIN {X 0,Y 445.038,Z 956.238,A -85,B 0,C 180,E1 17859.823,E2 17859.823} C_VEL
LIN {X 0,Y 452.312,Z 978.637,A -85,B 0,C 180,E1 17861.969,E2 17861.969} C_VEL
LIN {X 0,Y 444.375,Z 1022.833,A -85,B 0,C 180,E1 17864.092,E2 17864.092} C_VEL
LIN {X 0,Y 434.397,Z 1065.819,A -85,B 0,C 180,E1 17867.123,E2 17867.123} C_VEL
LIN {X 0,Y 423.667,Z 1104.571,A -85,B 0,C 180,E1 17870.922,E2 17870.922} C_VEL
LIN {X 0,Y 412.921,Z 1139.566,A -85,B 0,C 180,E1 17875.595,E2 17875.595} C_VEL
LIN {X 0,Y 403.855,Z 1169.815,A -85,B 0,C 180,E1 17881.12,E2 17881.12} C_VEL
LIN {X 0,Y 397.139,Z 1194.004,A -85,B 0,C 180,E1 17887.151,E2 17887.151} C_VEL
LIN {X 0,Y 392.91,Z 1212.695,A -85,B 0,C 180,E1 17893.763,E2 17893.763} C_VEL
LIN {X 0,Y 391.341,Z 1224.047,A -85,B 0,C 180,E1 17899.965,E2 17899.965} C_VEL
LIN {X 0,Y 390.847,Z 1229.721,A -85,B 0,C 180,E1 17905.553,E2 17905.553} C_VEL
LIN {X 0,Y 391.036,Z 1231.141,A -85,B 0,C 180,E1 17910,E2 17910} C_VEL
LIN {X 0,Y 390.877,Z 1229.728,A -85,B 0,C 180,E1 17914.446,E2 17914.446} C_VEL
LIN {X 0,Y 391.311,Z 1224.063,A -85,B 0,C 180,E1 17920.035,E2 17920.035} C_VEL
LIN {X 0,Y 392.939,Z 1212.724,A -85,B 0,C 180,E1 17926.235,E2 17926.235} C_VEL
LIN {X 0,Y 397.135,Z 1194.041,A -85,B 0,C 180,E1 17932.849,E2 17932.849} C_VEL
LIN {X 0,Y 403.846,Z 1169.873,A -85,B 0,C 180,E1 17938.881,E2 17938.881} C_VEL
LIN {X 0,Y 412.509,Z 1140.94,A -85,B 0,C 180,E1 17944.197,E2 17944.197} C_VEL
LIN {X 0,Y 422.692,Z 1107.947,A -85,B 0,C 180,E1 17948.69,E2 17948.69} C_VEL
LIN {X 0,Y 429.091,Z 1085.587,A -85,B 0,C 180,E1 17951.097,E2 17951.097} C_VEL
LIN {X 0,Y 429.425,Z 1072.552,A -85,B 0,C 180,E1 17952.673,E2 17952.673} C_VEL
LIN {X 0,Y 429.666,Z 1060.859,A -85,B 0,C 180,E1 17953.99,E2 17953.99} C_VEL
LIN {X 0,Y 430.116,Z 1059.011,A -85,B 0,C 180,E1 17954.139,E2 17954.139} C_VEL
LIN {X 0,Y 439.572,Z 1018.757,A -85,B 0,C 180,E1 17956.858,E2 17956.858} C_VEL
LIN {X 0,Y 446.654,Z 980.59,A -85,B 0,C 180,E1 17958.673,E2 17958.673} C_VEL
LIN {X 0,Y 435.443,Z 949.272,A -85,B 0,C 180,E1 17961.941,E2 17961.941} C_VEL
LIN {X 0,Y 419.779,Z 918.468,A -85,B 0,C 180,E1 17965.717,E2 17965.717} C_VEL
LIN {X 0,Y 402.219,Z 890.547,A -85,B 0,C 180,E1 17970.084,E2 17970.084} C_VEL
LIN {X 0,Y 389.048,Z 872.054,A -85,B 0,C 180,E1 17973.926,E2 17973.926} C_VEL
LIN {X 0,Y 384.891,Z 865.957,A -85,B 0,C 180,E1 17975.311,E2 17975.311} C_VEL
LIN {X 0,Y 381.541,Z 860.998,A -85,B 0,C 180,E1 17976.498,E2 17976.498} C_VEL
LIN {X 0,Y 381.392,Z 859.31,A -85,B 0,C 180,E1 17976.748,E2 17976.748} C_VEL
LIN {X 0,Y 381.684,Z 859.31,A -85,B 0,C 180,E1 17983.866,E2 17983.866} C_VEL
LIN {X 0,Y 382.172,Z 859.31,A -85,B 0,C 180,E1 17990.874,E2 17990.874} C_VEL
LIN {X 0,Y 382.74,Z 859.31,A -85,B 0,C 180,E1 17997.729,E2 17997.729} C_VEL
LIN {X 0,Y 382.793,Z 859.31,A -85,B 0,C 180,E1 18002.265,E2 18002.265} C_VEL
LIN {X 0,Y 382.184,Z 859.31,A -85,B 0,C 180,E1 18009.12,E2 18009.12} C_VEL
LIN {X 0,Y 381.704,Z 859.31,A -85,B 0,C 180,E1 18016.126,E2 18016.126} C_VEL
LIN {X 0,Y 381.311,Z 859.31,A -85,B 0,C 180,E1 18023.405,E2 18023.405} C_VEL
LIN {X 0,Y 380.979,Z 859.609,A -85,B 0,C 180,E1 18029.35,E2 18029.35} C_VEL
LIN {X 0,Y 383.027,Z 864.619,A -85,B 0,C 180,E1 18030.159,E2 18030.159} C_VEL
LIN {X 0,Y 386.276,Z 868.065,A -85,B 0,C 180,E1 18031.216,E2 18031.216} C_VEL
LIN {X 0,Y 404.134,Z 892.978,A -85,B 0,C 180,E1 18036.386,E2 18036.386} C_VEL
LIN {X 0,Y 424.15,Z 924.643,A -85,B 0,C 180,E1 18041.102,E2 18041.102} C_VEL
LIN {X 0,Y 442.232,Z 959.376,A -85,B 0,C 180,E1 18044.949,E2 18044.949} C_VEL
LIN {X 0,Y 449.061,Z 978.037,A -85,B 0,C 180,E1 18046.654,E2 18046.654} C_VEL
LIN {X 0,Y 441.893,Z 1020.483,A -85,B 0,C 180,E1 18048.283,E2 18048.283} C_VEL
LIN {X 0,Y 432.443,Z 1060.15,A -85,B 0,C 180,E1 18050.699,E2 18050.699} C_VEL
LIN {X 0,Y 421.866,Z 1095.484,A -85,B 0,C 180,E1 18053.817,E2 18053.817} C_VEL
LIN {X 0,Y 410.894,Z 1127.386,A -85,B 0,C 180,E1 18057.785,E2 18057.785} C_VEL
LIN {X 0,Y 401.284,Z 1153.199,A -85,B 0,C 180,E1 18062.21,E2 18062.21} C_VEL
LIN {X 0,Y 393.355,Z 1174.837,A -85,B 0,C 180,E1 18067.343,E2 18067.343} C_VEL
LIN {X 0,Y 387.272,Z 1192.88,A -85,B 0,C 180,E1 18073.54,E2 18073.54} C_VEL
LIN {X 0,Y 384.254,Z 1204.309,A -85,B 0,C 180,E1 18079.711,E2 18079.711} C_VEL
LIN {X 0,Y 383.218,Z 1210.014,A -85,B 0,C 180,E1 18085.464,E2 18085.464} C_VEL
LIN {X 0,Y 383.13,Z 1211.356,A -85,B 0,C 180,E1 18090,E2 18090} C_VEL
LIN {X 0,Y 383.228,Z 1209.937,A -85,B 0,C 180,E1 18094.536,E2 18094.536} C_VEL
LIN {X 0,Y 384.306,Z 1204.135,A -85,B 0,C 180,E1 18100.314,E2 18100.314} C_VEL
LIN {X 0,Y 387.358,Z 1192.586,A -85,B 0,C 180,E1 18106.481,E2 18106.481} C_VEL
LIN {X 0,Y 393.412,Z 1174.489,A -85,B 0,C 180,E1 18112.654,E2 18112.654} C_VEL
LIN {X 0,Y 402.094,Z 1151.058,A -85,B 0,C 180,E1 18118.104,E2 18118.104} C_VEL
LIN {X 0,Y 412.24,Z 1123.488,A -85,B 0,C 180,E1 18122.673,E2 18122.673} C_VEL
LIN {X 0,Y 422.894,Z 1092.13,A -85,B 0,C 180,E1 18126.423,E2 18126.423} C_VEL
LIN {X 0,Y 433.159,Z 1057.197,A -85,B 0,C 180,E1 18129.413,E2 18129.413} C_VEL
LIN {X 0,Y 442.05,Z 1019.053,A -85,B 0,C 180,E1 18131.685,E2 18131.685} C_VEL
LIN {X 0,Y 448.763,Z 979.138,A -85,B 0,C 180,E1 18133.221,E2 18133.221} C_VEL
LIN {X 0,Y 447.773,Z 973.231,A -85,B 0,C 180,E1 18133.608,E2 18133.608} C_VEL
LIN {X 0,Y 432.415,Z 939.562,A -85,B 0,C 180,E1 18137.03,E2 18137.03} C_VEL
LIN {X 0,Y 413.771,Z 907.846,A -85,B 0,C 180,E1 18141.095,E2 18141.095} C_VEL
LIN {X 0,Y 397.78,Z 884.212,A -85,B 0,C 180,E1 18145.166,E2 18145.166} C_VEL
LIN {X 0,Y 388.863,Z 872.047,A -85,B 0,C 180,E1 18147.78,E2 18147.78} C_VEL
LIN {X 0,Y 384.707,Z 866.025,A -85,B 0,C 180,E1 18149.141,E2 18149.141} C_VEL
LIN {X 0,Y 381.264,Z 861.411,A -85,B 0,C 180,E1 18150.322,E2 18150.322} C_VEL
LIN {X 0,Y 380.954,Z 859.31,A -85,B 0,C 180,E1 18150.577,E2 18150.577} C_VEL
LIN {X 0,Y 381.259,Z 859.31,A -85,B 0,C 180,E1 18156.591,E2 18156.591} C_VEL
LIN {X 0,Y 381.567,Z 859.31,A -85,B 0,C 180,E1 18163.868,E2 18163.868} C_VEL
LIN {X 0,Y 382.212,Z 859.31,A -85,B 0,C 180,E1 18170.881,E2 18170.881} C_VEL
LIN {X 0,Y 382.744,Z 859.31,A -85,B 0,C 180,E1 18177.735,E2 18177.735} C_VEL
LIN {X 0,Y 382.797,Z 859.31,A -85,B 0,C 180,E1 18182.271,E2 18182.271} C_VEL
LIN {X 0,Y 382.172,Z 859.31,A -85,B 0,C 180,E1 18189.126,E2 18189.126} C_VEL
LIN {X 0,Y 381.711,Z 859.31,A -85,B 0,C 180,E1 18196.133,E2 18196.133} C_VEL
LIN {X 0,Y 381.354,Z 859.543,A -85,B 0,C 180,E1 18203.461,E2 18203.461} C_VEL
LIN {X 0,Y 383.354,Z 864.657,A -85,B 0,C 180,E1 18204.27,E2 18204.27} C_VEL
LIN {X 0,Y 386.329,Z 867.729,A -85,B 0,C 180,E1 18205.232,E2 18205.232} C_VEL
LIN {X 0,Y 404.056,Z 893.202,A -85,B 0,C 180,E1 18210.453,E2 18210.453} C_VEL
LIN {X 0,Y 421.417,Z 921.604,A -85,B 0,C 180,E1 18214.722,E2 18214.722} C_VEL
LIN {X 0,Y 436.58,Z 952.413,A -85,B 0,C 180,E1 18218.417,E2 18218.417} C_VEL
LIN {X 0,Y 446.366,Z 979.873,A -85,B 0,C 180,E1 18221.269,E2 18221.269} C_VEL
LIN {X 0,Y 438.331,Z 1024.054,A -85,B 0,C 180,E1 18223.451,E2 18223.451} C_VEL
LIN {X 0,Y 428.351,Z 1065.748,A -85,B 0,C 180,E1 18226.422,E2 18226.422} C_VEL
LIN {X 0,Y 417.39,Z 1104.177,A -85,B 0,C 180,E1 18230.218,E2 18230.218} C_VEL
LIN {X 0,Y 406.605,Z 1138.176,A -85,B 0,C 180,E1 18234.78,E2 18234.78} C_VEL
LIN {X 0,Y 396.949,Z 1168.201,A -85,B 0,C 180,E1 18240.247,E2 18240.247} C_VEL
LIN {X 0,Y 389.901,Z 1192.637,A -85,B 0,C 180,E1 18246.358,E2 18246.358} C_VEL
LIN {X 0,Y 385.439,Z 1211.094,A -85,B 0,C 180,E1 18252.851,E2 18252.851} C_VEL
LIN {X 0,Y 383.69,Z 1222.182,A -85,B 0,C 180,E1 18258.611,E2 18258.611} C_VEL
LIN {X 0,Y 383.172,Z 1227.775,A -85,B 0,C 180,E1 18263.186,E2 18263.186} C_VEL
LIN {X 0,Y 383.077,Z 1230.579,A -85,B 0,C 180,E1 18267.733,E2 18267.733} C_VEL
LIN {X 0,Y 383.062,Z 1230.581,A -85,B 0,C 180,E1 18272.267,E2 18272.267} C_VEL
LIN {X 0,Y 383.266,Z 1225.667,A -85,B 0,C 180,E1 18278.811,E2 18278.811} C_VEL
LIN {X 0,Y 384.462,Z 1216.749,A -85,B 0,C 180,E1 18284.542,E2 18284.542} C_VEL
LIN {X 0,Y 387.729,Z 1200.512,A -85,B 0,C 180,E1 18291.192,E2 18291.192} C_VEL
LIN {X 0,Y 394.042,Z 1178.25,A -85,B 0,C 180,E1 18297.481,E2 18297.481} C_VEL
LIN {X 0,Y 403.039,Z 1149.536,A -85,B 0,C 180,E1 18303.356,E2 18303.356} C_VEL
LIN {X 0,Y 413.914,Z 1115.106,A -85,B 0,C 180,E1 18308.488,E2 18308.488} C_VEL
LIN {X 0,Y 425.331,Z 1077.019,A -85,B 0,C 180,E1 18312.601,E2 18312.601} C_VEL
LIN {X 0,Y 430.116,Z 1059.011,A -85,B 0,C 180,E1 18314.139,E2 18314.139} C_VEL
LIN {X 0,Y 431.155,Z 1048.388,A -85,B 0,C 180,E1 18315.158,E2 18315.158} C_VEL
LIN {X 0,Y 430.919,Z 1032.56,A -85,B 0,C 180,E1 18316.745,E2 18316.745} C_VEL
LIN {X 0,Y 431.264,Z 1030.637,A -85,B 0,C 180,E1 18316.878,E2 18316.878} C_VEL
LIN {X 0,Y 439.704,Z 989.616,A -85,B 0,C 180,E1 18319.034,E2 18319.034} C_VEL
LIN {X 0,Y 440.247,Z 981.702,A -85,B 0,C 180,E1 18319.472,E2 18319.472} C_VEL
LIN {X 0,Y 429.047,Z 950.606,A -85,B 0,C 180,E1 18322.872,E2 18322.872} C_VEL
LIN {X 0,Y 413.291,Z 919.581,A -85,B 0,C 180,E1 18326.878,E2 18326.878} C_VEL
LIN {X 0,Y 395.862,Z 892.159,A -85,B 0,C 180,E1 18331.479,E2 18331.479} C_VEL
LIN {X 0,Y 382.282,Z 872.91,A -85,B 0,C 180,E1 18335.773,E2 18335.773} C_VEL
LIN {X 0,Y 377.147,Z 865.888,A -85,B 0,C 180,E1 18337.642,E2 18337.642} C_VEL
LIN {X 0,Y 373.857,Z 861.121,A -85,B 0,C 180,E1 18338.956,E2 18338.956} C_VEL
LIN {X 0,Y 373.643,Z 859.31,A -85,B 0,C 180,E1 18339.205,E2 18339.205} C_VEL
LIN {X 0,Y 373.976,Z 859.31,A -85,B 0,C 180,E1 18346.517,E2 18346.517} C_VEL
LIN {X 0,Y 374.461,Z 859.31,A -85,B 0,C 180,E1 18353.026,E2 18353.026} C_VEL
LIN {X 0,Y 375.055,Z 859.31,A -85,B 0,C 180,E1 18359.997,E2 18359.997} C_VEL
LIN {X 0,Y 374.465,Z 859.31,A -85,B 0,C 180,E1 18366.968,E2 18366.968} C_VEL
LIN {X 0,Y 373.945,Z 859.31,A -85,B 0,C 180,E1 18374.064,E2 18374.064} C_VEL
LIN {X 0,Y 373.52,Z 859.31,A -85,B 0,C 180,E1 18381.405,E2 18381.405} C_VEL
LIN {X 0,Y 373.159,Z 859.77,A -85,B 0,C 180,E1 18386.811,E2 18386.811} C_VEL
LIN {X 0,Y 375.323,Z 864.827,A -85,B 0,C 180,E1 18387.772,E2 18387.772} C_VEL
LIN {X 0,Y 378.523,Z 867.923,A -85,B 0,C 180,E1 18388.928,E2 18388.928} C_VEL
LIN {X 0,Y 393.366,Z 888.544,A -85,B 0,C 180,E1 18393.776,E2 18393.776} C_VEL
LIN {X 0,Y 410.169,Z 913.726,A -85,B 0,C 180,E1 18398.233,E2 18398.233} C_VEL
LIN {X 0,Y 428.199,Z 944.82,A -85,B 0,C 180,E1 18402.318,E2 18402.318} C_VEL
LIN {X 0,Y 441.983,Z 975.783,A -85,B 0,C 180,E1 18405.591,E2 18405.591} C_VEL
LIN {X 0,Y 443.235,Z 980.878,A -85,B 0,C 180,E1 18406.004,E2 18406.004} C_VEL
LIN {X 0,Y 436.073,Z 1021.256,A -85,B 0,C 180,E1 18407.597,E2 18407.597} C_VEL
LIN {X 0,Y 426.928,Z 1058.822,A -85,B 0,C 180,E1 18409.888,E2 18409.888} C_VEL
LIN {X 0,Y 416.34,Z 1093.591,A -85,B 0,C 180,E1 18412.931,E2 18412.931} C_VEL
LIN {X 0,Y 405.075,Z 1125.376,A -85,B 0,C 180,E1 18416.833,E2 18416.833} C_VEL
LIN {X 0,Y 394.361,Z 1153.17,A -85,B 0,C 180,E1 18421.609,E2 18421.609} C_VEL
LIN {X 0,Y 385.981,Z 1175.068,A -85,B 0,C 180,E1 18426.885,E2 18426.885} C_VEL
LIN {X 0,Y 380.091,Z 1191.511,A -85,B 0,C 180,E1 18432.507,E2 18432.507} C_VEL
LIN {X 0,Y 376.784,Z 1202.935,A -85,B 0,C 180,E1 18438.4,E2 18438.4} C_VEL
LIN {X 0,Y 375.586,Z 1208.506,A -85,B 0,C 180,E1 18443.049,E2 18443.049} C_VEL
LIN {X 0,Y 375.203,Z 1211.236,A -85,B 0,C 180,E1 18447.686,E2 18447.686} C_VEL
LIN {X 0,Y 375.259,Z 1211.19,A -85,B 0,C 180,E1 18452.315,E2 18452.315} C_VEL
LIN {X 0,Y 375.871,Z 1207.253,A -85,B 0,C 180,E1 18458.112,E2 18458.112} C_VEL
LIN {X 0,Y 378.192,Z 1197.728,A -85,B 0,C 180,E1 18464.503,E2 18464.503} C_VEL
LIN {X 0,Y 383.297,Z 1182.102,A -85,B 0,C 180,E1 18470.843,E2 18470.843} C_VEL
LIN {X 0,Y 391.518,Z 1160.398,A -85,B 0,C 180,E1 18476.739,E2 18476.739} C_VEL
LIN {X 0,Y 401.969,Z 1133.313,A -85,B 0,C 180,E1 18481.854,E2 18481.854} C_VEL
LIN {X 0,Y 412.998,Z 1102.953,A -85,B 0,C 180,E1 18485.948,E2 18485.948} C_VEL
LIN {X 0,Y 423.843,Z 1069.036,A -85,B 0,C 180,E1 18489.224,E2 18489.224} C_VEL
LIN {X 0,Y 433.871,Z 1030.429,A -85,B 0,C 180,E1 18491.825,E2 18491.825} C_VEL
LIN {X 0,Y 441.537,Z 991.069,A -85,B 0,C 180,E1 18493.568,E2 18493.568} C_VEL
LIN {X 0,Y 442.777,Z 978.137,A -85,B 0,C 180,E1 18494.075,E2 18494.075} C_VEL
LIN {X 0,Y 428.066,Z 944.709,A -85,B 0,C 180,E1 18497.58,E2 18497.58} C_VEL
LIN {X 0,Y 409.882,Z 913.28,A -85,B 0,C 180,E1 18501.702,E2 18501.702} C_VEL
LIN {X 0,Y 392.152,Z 886.573,A -85,B 0,C 180,E1 18506.438,E2 18506.438} C_VEL
LIN {X 0,Y 381.475,Z 872.395,A -85,B 0,C 180,E1 18509.832,E2 18509.832} C_VEL
LIN {X 0,Y 377.269,Z 866.253,A -85,B 0,C 180,E1 18511.356,E2 18511.356} C_VEL
LIN {X 0,Y 373.505,Z 861.758,A -85,B 0,C 180,E1 18512.797,E2 18512.797} C_VEL
LIN {X 0,Y 373.123,Z 859.31,A -85,B 0,C 180,E1 18513.083,E2 18513.083} C_VEL
LIN {X 0,Y 373.476,Z 859.31,A -85,B 0,C 180,E1 18518.936,E2 18518.936} C_VEL
LIN {X 0,Y 373.899,Z 859.31,A -85,B 0,C 180,E1 18526.568,E2 18526.568} C_VEL
LIN {X 0,Y 374.486,Z 859.31,A -85,B 0,C 180,E1 18533.033,E2 18533.033} C_VEL
LIN {X 0,Y 375.06,Z 859.31,A -85,B 0,C 180,E1 18540.003,E2 18540.003} C_VEL
LIN {X 0,Y 374.461,Z 859.31,A -85,B 0,C 180,E1 18546.974,E2 18546.974} C_VEL
LIN {X 0,Y 373.943,Z 859.31,A -85,B 0,C 180,E1 18554.071,E2 18554.071} C_VEL
LIN {X 0,Y 373.637,Z 859.929,A -85,B 0,C 180,E1 18561.001,E2 18561.001} C_VEL
LIN {X 0,Y 375.848,Z 864.954,A -85,B 0,C 180,E1 18561.972,E2 18561.972} C_VEL
LIN {X 0,Y 378.902,Z 868.161,A -85,B 0,C 180,E1 18563.087,E2 18563.087} C_VEL
LIN {X 0,Y 393.35,Z 888.668,A -85,B 0,C 180,E1 18567.853,E2 18567.853} C_VEL
LIN {X 0,Y 410.614,Z 915.073,A -85,B 0,C 180,E1 18572.501,E2 18572.501} C_VEL
LIN {X 0,Y 427.656,Z 947.741,A -85,B 0,C 180,E1 18576.793,E2 18576.793} C_VEL
LIN {X 0,Y 439.455,Z 979.155,A -85,B 0,C 180,E1 18580.279,E2 18580.279} C_VEL
LIN {X 0,Y 440.217,Z 985.164,A -85,B 0,C 180,E1 18580.775,E2 18580.775} C_VEL
LIN {X 0,Y 432.093,Z 1026.44,A -85,B 0,C 180,E1 18582.867,E2 18582.867} C_VEL
LIN {X 0,Y 422.111,Z 1066.564,A -85,B 0,C 180,E1 18585.778,E2 18585.778} C_VEL
LIN {X 0,Y 410.749,Z 1105.021,A -85,B 0,C 180,E1 18589.641,E2 18589.641} C_VEL
LIN {X 0,Y 399.471,Z 1139.278,A -85,B 0,C 180,E1 18594.334,E2 18594.334} C_VEL
LIN {X 0,Y 389.417,Z 1169.228,A -85,B 0,C 180,E1 18599.934,E2 18599.934} C_VEL
LIN {X 0,Y 382.199,Z 1193.199,A -85,B 0,C 180,E1 18606.102,E2 18606.102} C_VEL
LIN {X 0,Y 377.416,Z 1212.248,A -85,B 0,C 180,E1 18613.077,E2 18613.077} C_VEL
LIN {X 0,Y 375.609,Z 1223.622,A -85,B 0,C 180,E1 18619.54,E2 18619.54} C_VEL
LIN {X 0,Y 375.05,Z 1229.315,A -85,B 0,C 180,E1 18625.365,E2 18625.365} C_VEL
LIN {X 0,Y 375.238,Z 1230.737,A -85,B 0,C 180,E1 18630,E2 18630} C_VEL
LIN {X 0,Y 375.075,Z 1229.323,A -85,B 0,C 180,E1 18634.634,E2 18634.634} C_VEL
LIN {X 0,Y 375.582,Z 1223.641,A -85,B 0,C 180,E1 18640.46,E2 18640.46} C_VEL
LIN {X 0,Y 377.447,Z 1212.282,A -85,B 0,C 180,E1 18646.921,E2 18646.921} C_VEL
LIN {X 0,Y 382.188,Z 1193.251,A -85,B 0,C 180,E1 18653.897,E2 18653.897} C_VEL
LIN {X 0,Y 389.497,Z 1169.303,A -85,B 0,C 180,E1 18660.058,E2 18660.058} C_VEL
LIN {X 0,Y 399.523,Z 1139.354,A -85,B 0,C 180,E1 18665.666,E2 18665.666} C_VEL
LIN {X 0,Y 411.069,Z 1104.03,A -85,B 0,C 180,E1 18670.502,E2 18670.502} C_VEL
LIN {X 0,Y 422.701,Z 1064.703,A -85,B 0,C 180,E1 18674.401,E2 18674.401} C_VEL
LIN {X 0,Y 431.264,Z 1030.637,A -85,B 0,C 180,E1 18676.878,E2 18676.878} C_VEL
LIN {X 0,Y 431.72,Z 1015.848,A -85,B 0,C 180,E1 18678.133,E2 18678.133} C_VEL
LIN {X 0,Y 432.113,Z 1000.704,A -85,B 0,C 180,E1 18679.291,E2 18679.291} C_VEL
LIN {X 0,Y 434.686,Z 985.606,A -85,B 0,C 180,E1 18680,E2 18680} C_VEL
LIN {X 0,Y 423.774,Z 954.402,A -85,B 0,C 180,E1 18683.534,E2 18683.534} C_VEL
LIN {X 0,Y 408.81,Z 924.332,A -85,B 0,C 180,E1 18687.574,E2 18687.574} C_VEL
LIN {X 0,Y 392.628,Z 898.441,A -85,B 0,C 180,E1 18692.025,E2 18692.025} C_VEL
LIN {X 0,Y 379.392,Z 879.539,A -85,B 0,C 180,E1 18696.345,E2 18696.345} C_VEL
LIN {X 0,Y 374.427,Z 872.727,A -85,B 0,C 180,E1 18698.214,E2 18698.214} C_VEL
LIN {X 0,Y 370.239,Z 866.472,A -85,B 0,C 180,E1 18699.975,E2 18699.975} C_VEL
LIN {X 0,Y 366.132,Z 861.835,A -85,B 0,C 180,E1 18701.785,E2 18701.785} C_VEL
LIN {X 0,Y 365.721,Z 859.31,A -85,B 0,C 180,E1 18702.288,E2 18702.288} C_VEL
LIN {X 0,Y 366.133,Z 859.31,A -85,B 0,C 180,E1 18708.057,E2 18708.057} C_VEL
LIN {X 0,Y 366.773,Z 859.31,A -85,B 0,C 180,E1 18715.258,E2 18715.258} C_VEL
LIN {X 0,Y 367.152,Z 859.31,A -85,B 0,C 180,E1 18719.997,E2 18719.997} C_VEL
LIN {X 0,Y 366.537,Z 859.31,A -85,B 0,C 180,E1 18727.173,E2 18727.173} C_VEL
LIN {X 0,Y 365.984,Z 859.31,A -85,B 0,C 180,E1 18734.377,E2 18734.377} C_VEL
LIN {X 0,Y 365.535,Z 859.31,A -85,B 0,C 180,E1 18741.896,E2 18741.896} C_VEL
LIN {X 0,Y 365.502,Z 859.654,A -85,B 0,C 180,E1 18743.908,E2 18743.908} C_VEL
LIN {X 0,Y 367.281,Z 864.521,A -85,B 0,C 180,E1 18744.867,E2 18744.867} C_VEL
LIN {X 0,Y 370.864,Z 867.882,A -85,B 0,C 180,E1 18746.369,E2 18746.369} C_VEL
LIN {X 0,Y 375.12,Z 873.565,A -85,B 0,C 180,E1 18748.078,E2 18748.078} C_VEL
LIN {X 0,Y 390.41,Z 894.935,A -85,B 0,C 180,E1 18753.255,E2 18753.255} C_VEL
LIN {X 0,Y 407.785,Z 921.401,A -85,B 0,C 180,E1 18757.973,E2 18757.973} C_VEL
LIN {X 0,Y 425.149,Z 952.552,A -85,B 0,C 180,E1 18762.065,E2 18762.065} C_VEL
LIN {X 0,Y 437.499,Z 982.23,A -85,B 0,C 180,E1 18765.276,E2 18765.276} C_VEL
LIN {X 0,Y 430.254,Z 1022.261,A -85,B 0,C 180,E1 18766.905,E2 18766.905} C_VEL
LIN {X 0,Y 420.88,Z 1059.458,A -85,B 0,C 180,E1 18769.204,E2 18769.204} C_VEL
LIN {X 0,Y 409.638,Z 1095.102,A -85,B 0,C 180,E1 18772.385,E2 18772.385} C_VEL
LIN {X 0,Y 398.237,Z 1126.194,A -85,B 0,C 180,E1 18776.286,E2 18776.286} C_VEL
LIN {X 0,Y 387.344,Z 1153.427,A -85,B 0,C 180,E1 18781.046,E2 18781.046} C_VEL
LIN {X 0,Y 378.205,Z 1176.334,A -85,B 0,C 180,E1 18786.726,E2 18786.726} C_VEL
LIN {X 0,Y 371.893,Z 1193.55,A -85,B 0,C 180,E1 18792.953,E2 18792.953} C_VEL
LIN {X 0,Y 368.58,Z 1204.807,A -85,B 0,C 180,E1 18799.339,E2 18799.339} C_VEL
LIN {X 0,Y 367.442,Z 1210.421,A -85,B 0,C 180,E1 18805.269,E2 18805.269} C_VEL
LIN {X 0,Y 367.333,Z 1211.76,A -85,B 0,C 180,E1 18810,E2 18810} C_VEL
LIN {X 0,Y 367.454,Z 1210.344,A -85,B 0,C 180,E1 18814.731,E2 18814.731} C_VEL
LIN {X 0,Y 368.637,Z 1204.67,A -85,B 0,C 180,E1 18820.66,E2 18820.66} C_VEL
LIN {X 0,Y 371.986,Z 1193.23,A -85,B 0,C 180,E1 18827.083,E2 18827.083} C_VEL
LIN {X 0,Y 377.9,Z 1176.905,A -85,B 0,C 180,E1 18832.994,E2 18832.994} C_VEL
LIN {X 0,Y 386.459,Z 1155.537,A -85,B 0,C 180,E1 18838.387,E2 18838.387} C_VEL
LIN {X 0,Y 396.398,Z 1130.552,A -85,B 0,C 180,E1 18842.941,E2 18842.941} C_VEL
LIN {X 0,Y 407.54,Z 1100.6,A -85,B 0,C 180,E1 18846.91,E2 18846.91} C_VEL
LIN {X 0,Y 418.646,Z 1066.535,A -85,B 0,C 180,E1 18850.145,E2 18850.145} C_VEL
LIN {X 0,Y 428.49,Z 1029.337,A -85,B 0,C 180,E1 18852.622,E2 18852.622} C_VEL
LIN {X 0,Y 436.365,Z 989.298,A -85,B 0,C 180,E1 18854.379,E2 18854.379} C_VEL
LIN {X 0,Y 437.019,Z 981.044,A -85,B 0,C 180,E1 18854.737,E2 18854.737} C_VEL
LIN {X 0,Y 422.893,Z 948.153,A -85,B 0,C 180,E1 18858.337,E2 18858.337} C_VEL
LIN {X 0,Y 404.778,Z 916.577,A -85,B 0,C 180,E1 18862.641,E2 18862.641} C_VEL
LIN {X 0,Y 388.496,Z 892.3,A -85,B 0,C 180,E1 18867.166,E2 18867.166} C_VEL
LIN {X 0,Y 378.66,Z 878.971,A -85,B 0,C 180,E1 18870.411,E2 18870.411} C_VEL
LIN {X 0,Y 374.345,Z 872.997,A -85,B 0,C 180,E1 18872.023,E2 18872.023} C_VEL
LIN {X 0,Y 370.686,Z 867.376,A -85,B 0,C 180,E1 18873.535,E2 18873.535} C_VEL
LIN {X 0,Y 365.877,Z 862.122,A -85,B 0,C 180,E1 18875.602,E2 18875.602} C_VEL
LIN {X 0,Y 365.43,Z 859.31,A -85,B 0,C 180,E1 18876.035,E2 18876.035} C_VEL
LIN {X 0,Y 365.683,Z 859.31,A -85,B 0,C 180,E1 18883.146,E2 18883.146} C_VEL
LIN {X 0,Y 366.318,Z 859.31,A -85,B 0,C 180,E1 18890.482,E2 18890.482} C_VEL
LIN {X 0,Y 366.925,Z 859.31,A -85,B 0,C 180,E1 18897.637,E2 18897.637} C_VEL
LIN {X 0,Y 366.971,Z 859.31,A -85,B 0,C 180,E1 18902.369,E2 18902.369} C_VEL
LIN {X 0,Y 366.292,Z 859.31,A -85,B 0,C 180,E1 18909.525,E2 18909.525} C_VEL
LIN {X 0,Y 365.818,Z 859.31,A -85,B 0,C 180,E1 18916.854,E2 18916.854} C_VEL
LIN {X 0,Y 365.744,Z 859.486,A -85,B 0,C 180,E1 18918.032,E2 18918.032} C_VEL
LIN {X 0,Y 367.58,Z 864.352,A -85,B 0,C 180,E1 18919.024,E2 18919.024} C_VEL
LIN {X 0,Y 371.236,Z 867.897,A -85,B 0,C 180,E1 18920.554,E2 18920.554} C_VEL
LIN {X 0,Y 375.428,Z 873.589,A -85,B 0,C 180,E1 18922.232,E2 18922.232} C_VEL
LIN {X 0,Y 390.998,Z 896.214,A -85,B 0,C 180,E1 18927.553,E2 18927.553} C_VEL
LIN {X 0,Y 407.119,Z 921.343,A -85,B 0,C 180,E1 18932.025,E2 18932.025} C_VEL
LIN {X 0,Y 423.018,Z 953,A -85,B 0,C 180,E1 18936.303,E2 18936.303} C_VEL
LIN {X 0,Y 434.111,Z 983.883,A -85,B 0,C 180,E1 18939.832,E2 18939.832} C_VEL
LIN {X 0,Y 433.779,Z 991.161,A -85,B 0,C 180,E1 18940.268,E2 18940.268} C_VEL
LIN {X 0,Y 424.734,Z 1033.725,A -85,B 0,C 180,E1 18942.573,E2 18942.573} C_VEL
LIN {X 0,Y 414.235,Z 1073.088,A -85,B 0,C 180,E1 18945.622,E2 18945.622} C_VEL
LIN {X 0,Y 403.19,Z 1108.587,A -85,B 0,C 180,E1 18949.375,E2 18949.375} C_VEL
LIN {X 0,Y 392.259,Z 1140.565,A -85,B 0,C 180,E1 18953.907,E2 18953.907} C_VEL
LIN {X 0,Y 382.346,Z 1168.957,A -85,B 0,C 180,E1 18959.319,E2 18959.319} C_VEL
LIN {X 0,Y 374.72,Z 1192.948,A -85,B 0,C 180,E1 18965.594,E2 18965.594} C_VEL
LIN {X 0,Y 369.678,Z 1212.025,A -85,B 0,C 180,E1 18972.712,E2 18972.712} C_VEL
LIN {X 0,Y 367.759,Z 1223.41,A -85,B 0,C 180,E1 18979.314,E2 18979.314} C_VEL
